(* CoDeSys 2.3 project: cy-wg-019-003.pro *)
(* Title: cy-wg-06 - ClevergyAS *)
(* Author: Andrea Ravasio *)
(* Libraries: Standard.lib 2.12.10 13:48:34, Util.lib 26.9.14 09:12:46, Visual.lib 2.12.10 13:48:34, WagoLibIdent.lib 25.2.13 10:12:16, WagoLibStatus.lib 2.12.10 13:48:32, SysLibFile.lib 2.12.10 13:48:34, SysLibRtc.lib 2.12.10 13:48:32, SysLibSockets.lib 10.2.11 08:20:54, SysLibEvent.lib 2.12.10 13:48:34, SysLibPlcCtrl.lib 2.12.10 13:48:32, SysLibCallback.lib 2.12.10 13:48:32, mod_com.lib 2.12.10 13:48:32, SerComm.lib 31.5.11 07:54:36, Serial_Interface_01.lib 22.4.13 11:50:14, Modb_l05.lib 13.5.15 09:30:08, Ethernet.lib 2.12.10 13:48:32, MBus_03.lib 9.2.13 16:51:58, WagoLibModbus_IP_01.lib 24.7.13 14:05:58, WagoLibMBX_01.lib 20.3.12 15:32:40, LON_01.lib 28.9.12 13:05:10 *)

(* PLC configuration (modules and I/O channels)
VPN_ST2 AT %IX28.0 [BOOLOnX_I] Ch_1 Digital input
LAMP_AL AT %QX18.0 [BOOLOnX_Q] Ch_1 Digital output
KEY_QE_ST AT %IX28.1 [BOOLOnX_I] Ch_2 Digital input
CIR02_EN AT %QX18.1 [BOOLOnX_Q] Ch_2 Digital output
ALARM_PB AT %IX28.2 [BOOLOnX_I] Ch_3 Digital input
CIR01_EN AT %QX18.2 [BOOLOnX_Q] Ch_3 Digital output
CIRD02_A_AL AT %IX28.3 [BOOLOnX_I] Ch_4 Digital input
CIR03_EN AT %QX18.3 [BOOLOnX_Q] Ch_4 Digital output
CIRD02_A_AUTO AT %IX28.4 [BOOLOnX_I] Ch_5 Digital input
AT %QX18.4 [BOOLOnX_Q] Ch_5 Digital output
CIRD02_B_AL AT %IX28.5 [BOOLOnX_I] Ch_6 Digital input
AT %QX18.5 [BOOLOnX_Q] Ch_6 Digital output
CIRD02_B_AUTO AT %IX28.6 [BOOLOnX_I] Ch_7 Digital input
AT %QX18.6 [BOOLOnX_Q] Ch_7 Digital output
CIRD03_A_AL AT %IX28.7 [BOOLOnX_I] Ch_8 Digital input
AT %QX18.7 [BOOLOnX_Q] Ch_8 Digital output
0750-9999/0400-0008 8 DI Generic [Type_1_8_Channels] node 1, in %IB56 out %QB36 {INTTypePAAssignment = PLC; INTTypeModule = plugged}
  CIRD01_B_AUTO AT %IX28.8 [BOOLOnX_I] I 1: Digital Input
  CIR02_ST AT %IX28.9 [BOOLOnX_I] I 2: Digital Input
  CIRD01_A_AL AT %IX28.10 [BOOLOnX_I] I 3: Digital Input
  CIR02_AUTO AT %IX28.11 [BOOLOnX_I] I 4: Digital Input
  CIRD01_A_AUTO AT %IX28.12 [BOOLOnX_I] I 5: Digital Input
  CIR01_AL AT %IX28.13 [BOOLOnX_I] I 6: Digital Input
  CIR02_AL AT %IX28.14 [BOOLOnX_I] I 7: Digital Input
  CIR01_ST AT %IX28.15 [BOOLOnX_I] I 8: Digital Input
0750-9999/0400-0008 8 DI Generic [Type_1_8_Channels] node 2, in %IB57 out %QB37 {INTTypePAAssignment = PLC; INTTypeModule = plugged}
  CIR01_AUTO AT %IX29.0 [BOOLOnX_I] I 1: Digital Input
  CTL03_ST AT %IX29.1 [BOOLOnX_I] I 2: Digital Input
  CIR03_AL AT %IX29.2 [BOOLOnX_I] I 3: Digital Input
  CTL01_ST AT %IX29.3 [BOOLOnX_I] I 4: Digital Input
  CIR03_ST AT %IX29.4 [BOOLOnX_I] I 5: Digital Input
  CTL02_ST AT %IX29.5 [BOOLOnX_I] I 6: Digital Input
  CIR03_AUTO AT %IX29.6 [BOOLOnX_I] I 7: Digital Input
  CIRD01_B_AL AT %IX29.7 [BOOLOnX_I] I 8: Digital Input
0750-9999/0400-0004 4 DI Generic [Type_1_4_Channels] node 3, in %IB58 out %QB37 {INTTypePAAssignment = PLC; INTTypeModule = plugged}
  CIRD03_A_AUTO AT %IX29.8 [BOOLOnX_I] I 1: Digital Input
  CIRD03_B_AUTO AT %IX29.9 [BOOLOnX_I] I 2: Digital Input
  CIRD03_B_AL AT %IX29.10 [BOOLOnX_I] I 3: Digital Input
  AT %IX29.11 [BOOLOnX_I] I 4: Digital Input
0753-0648 LON-FTT [Type_55_1_Channels] node 4, in %IB52 out %QB36 {INTTypePAAssignment = PLC; INTTypeModule = plugged; DataStream = .; DataStream = .; DataStream = .; DataStream = .; DataStream = .; DataStream = .; DataStream = .; DataStream = .; DataStream = .; DataStream = .; DataStream = .; DataStream = .; DataStream = .; DataStream = .; DataStream = .; DataStream = .; DataStream = .; DataStream = .; DataStream = .; DataStream = .; DataStream = .; DataStream = .; DataStream = .; DataStream = .; DataStream = .; DataStream = .; DataStream = .; DataStream = .; DataStream = .; DataStream = .; DataStream = .; DataStream = .; DataStream = .; DataStream = .; DataStream = .; DataStream = .; DataStream = .; DataStream = .; DataStream = .; DataStream = .; DataStream = .; DataStream = .; DataStream = .; DataStream = .; DataStream = .; DataStream = .; DataStream = .; DataStream = .; DataStream = .; DataStream = .; DataStream = .; DataStream = .; DataStream = .; DataStream = .; DataStream = .; DataStream = .; DataStream = .; DataStream = .; DataStream = .; DataStream = .; DataStream = .; DataStream = .; DataStream = .; DataStream = .; DataStream = .; DataStream = .; DataStream = .; DataStream = .; DataStream = .; DataStream = .; DataStream = .; DataStream = .; DataStream = .; DataStream = .; DataStream = .; DataStream = .; DataStream = .; DataStream = .; DataStream = .; DataStream = .; DataStream = .; DataStream = .; DataStream = .; DataStream = .; DataStream = .; DataStream = .; DataStream = .; DataStream = .; DataStream = .; DataStream = .; DataStream = .; DataStream = .; DataStream = .; DataStream = .; DataStream = .; DataStream = .; DataStream = .; DataStream = .; DataStream = .; DataStream = .; DataStream = .; DataStream = .; DataStream = .; DataStream = .; DataStream = .; DataStream = .; DataStream = .; DataStream = .; DataStream = .; DataStream = .; DataStream = .; DataStream = .; DataStream = .; DataStream = .; DataStream = .; DataStream = .; DataStream = .; DataStream = .; DataStream = .; DataStream = .; DataStream = .; DataStream = .; DataStream = .; DataStream = .; DataStream = .; DataStream = .; DataStream = .; DataStream = .; DataStream = .; DataStream = .; DataStream = .; DataStream = .; DataStream = .; DataStream = .; DataStream = .; DataStream = .; DataStream = .; DataStream = .; DataStream = .; DataStream = .; DataStream = .; DataStream = .; DataStream = .; DataStream = .; DataStream = .; DataStream = .; DataStream = .; DataStream = .; DataStream = .; DataStream = .; DataStream = .; DataStream = .; DataStream = .; DataStream = .; DataStream = .; DataStream = .; DataStream = .; DataStream = .; DataStream = .; DataStream = .; DataStream = .; DataStream = .; DataStream = .; DataStream = .; DataStream = .; DataStream = .; DataStream = .; DataStream = .; DataStream = .; DataStream = .; DataStream = .; DataStream = .; DataStream = .; DataStream = .; DataStream = .; DataStream = .; DataStream = .; DataStream = .; DataStream = .; DataStream = .; DataStream = .; DataStream = .; DataStream = .; DataStream = .; DataStream = .; DataStream = .; DataStream = .; DataStream = .; DataStream = .; DataStream = .; DataStream = .; DataStream = .; DataStream = .; DataStream = .; DataStream = .; DataStream = .; DataStream = .; DataStream = .; DataStream = .; DataStream = .}
  AT %IB0 [BYTEOnB_I] First Byte of 24
  AT %QB0 [BYTEOnB_Q] First Byte of 24
0750-0464#04 2/4 AI RTD / ADJ./ HA [Type_44_4_Channels] node 5, in %IB52 out %QB36 {INTTypePAAssignment = PLC; INTTypeModule = plugged}
  S01 AT %IW12 [INTOnW_I] Channel 1
  S02 AT %IW13 [INTOnW_I] Channel 2
  S03 AT %IW14 [INTOnW_I] Channel 3
  S04 AT %IW15 [INTOnW_I] Channel 4
  S05 AT %IW16 [INTOnW_I] Channel 1
  AT %IW17 [INTOnW_I] Channel 2
  S12 AT %IW18 [INTOnW_I] Channel 3
  AT %IW19 [INTOnW_I] Channel 4
0750-0478 2 AI 0-10V 16 Bit S.E. [Type_8_2_Channels] node 7, in %IB84 out %QB60 {INTTypePAAssignment = PLC; INTTypeModule = plugged}
  VRD02_ST AT %IW20 [WORDOnW_I] I 1: Analog Input
  AT %IW21 [WORDOnW_I] I 2: Analog Input
0750-0556 2 AO ±10V [Type_14_2_Channels] node 8, in %IB92 out %QB60 {INTTypePAAssignment = PLC; INTTypeModule = plugged}
  VRD02_CTRL AT %QW12 [WORDOnW_Q] O 1: Analog Output
  AT %QW13 [WORDOnW_Q] O 2: Analog Output
0750-0650/0003-0000#03 RS 232 C Interface (Adjustable), 3 Byte [Type_21_1_Channels] node 9, in %IB96 out %QB60 {INTTypePAAssignment = PLC; INTTypeModule = plugged}
  AT %IX22.0 [BOOLOnX_I] Transmission acknowledgement
  AT %IX22.1 [BOOLOnX_I] Reception request
  AT %IX22.2 [BOOLOnX_I] Initialization acknowledgement
  AT %IX22.3 [BOOLOnX_I] Input buffer is full
  AT %IX22.4 [BOOLOnX_I] Number of received characters Bit 0
  AT %IX22.5 [BOOLOnX_I] Number of received characters Bit 1
  AT %IX22.6 [BOOLOnX_I] Number of received characters Bit 2
  AT %IB45 [BYTEOnB_I] Input data Byte 0
  AT %IB46 [BYTEOnB_I] Input data Byte 1
  AT %IB47 [BYTEOnB_I] Input data Byte 2
  AT %QX14.0 [BOOLOnX_Q] Transmission request
  AT %QX14.1 [BOOLOnX_Q] Reception acknowledgement
  AT %QX14.2 [BOOLOnX_Q] Initialization request
  AT %QX14.4 [BOOLOnX_Q] Number of characters Bit 0
  AT %QX14.5 [BOOLOnX_Q] Number of characters Bit 1
  AT %QX14.6 [BOOLOnX_Q] Number of characters Bit 2
  AT %QB29 [BYTEOnB_Q] Output data Byte 0
  AT %QB30 [BYTEOnB_Q] Output data Byte 1
  AT %QB31 [BYTEOnB_Q] Output data Byte 2
0750-0653/0003-0000#03 RS485 Interface (Adjustable), 3 Bytes [Type_21_1_Channels] node 10, in %IB96 out %QB64 {INTTypePAAssignment = PLC; INTTypeModule = plugged}
  AT %IX24.0 [BOOLOnX_I] Transmission acknowledgement
  AT %IX24.1 [BOOLOnX_I] Reception request
  AT %IX24.2 [BOOLOnX_I] Initialization acknowledgement
  AT %IX24.3 [BOOLOnX_I] Input buffer is full
  AT %IX24.4 [BOOLOnX_I] Number of received characters Bit 0
  AT %IX24.5 [BOOLOnX_I] Number of received characters Bit 1
  AT %IX24.6 [BOOLOnX_I] Number of received characters Bit 2
  AT %IB49 [BYTEOnB_I] Input data Byte 0
  AT %IB50 [BYTEOnB_I] Input data Byte 1
  AT %IB51 [BYTEOnB_I] Input data Byte 2
  AT %QX16.0 [BOOLOnX_Q] Transmission request
  AT %QX16.1 [BOOLOnX_Q] Reception acknowledgement
  AT %QX16.2 [BOOLOnX_Q] Initialization request
  AT %QX16.4 [BOOLOnX_Q] Number of characters Bit 0
  AT %QX16.5 [BOOLOnX_Q] Number of characters Bit 1
  AT %QX16.6 [BOOLOnX_Q] Number of characters Bit 2
  AT %QB33 [BYTEOnB_Q] Output data Byte 0
  AT %QB34 [BYTEOnB_Q] Output data Byte 1
  AT %QB35 [BYTEOnB_Q] Output data Byte 2
0750-0461/0000-0007 2 AI PT100 Resistor Measur. 10R-5k0 [Type_8_2_Channels] node 11, in %IB100 out %QB68 {INTTypePAAssignment = PLC; INTTypeModule = plugged}
  VRD01_ST AT %IW26 [WORDOnW_I] I 1: Analog Input
  AT %IW27 [WORDOnW_I] I 2: Analog Input
VRD01_OP AT %QX18.8 [BOOLOnX_Q] O 1: Digital Output
VRD01_CL AT %QX18.9 [BOOLOnX_Q] O 2: Digital Output
CIRD01_B_EN AT %QX18.10 [BOOLOnX_Q] O 1: Digital Output
CIRD01_A_EN AT %QX18.11 [BOOLOnX_Q] O 2: Digital Output
Fieldbus variables [FB_VARS] node 1, in %IB0 out %QB0
Flag variables [FLAG_VARS] node 2, in %IB0 out %QB0
Modbus-Master [MB_MASTER] node 3, in %IB0 out %QB0
*)

(* Global variable list: Global_Constants *)
VAR_GLOBAL CONSTANT

	Plant_NAME			: STRING :='cySN:19 cyVER:1 - ';
	Plant_SN			: DWORD  :=19;	(* S/N Impianto di telecontrollo *)
	Plant_SW_VER		: WORD   :=1;		(* Versione SW installata *)


	(* Colour defines *)
	COLOR_RED			: DWORD	:= 16#2020F0;
	COLOR_YELLOW		: DWORD	:= 16#20F0F0;
	COLOR_GREEN			: DWORD	:= 16#20F020;
	COLOR_LIGHT_GREEN	: DWORD := 16#006000;

	(* Parameters *)
	Plant_DefaultTAmb	: INT	:=100;		(* [.1°C] Temperatura ambiente di default in caso di rottura sonda *)
	Plant_MaxRunTAmb	: INT   :=210; 		(* [.1°C] Temperatura ambiente massima funzionamento impianto *)
	Plant_AntiFreezeTAmb: INT   :=-40;		(* [.1°C] Antifreeze temperature, start circulators *)
	Plant_VRD_TAlarm	: INT   :=850; 		(* [.1°C] Temperatura di allarme VRD, blocco *)
	Plant_VRD_TMax		: INT   :=800; 		(* [.1°C] Setpoint massimo per uscita VRD *)
	Plant_VRD_TDefault	: INT	:=300;		(* [.1°C] Temperatura di default in caso di errore climatica *)
	Plant_CirOffDelay	: TIME	:=T#30m;	(* (Def.T#15m) Ritardo spegnimento pompe per ricircolo caldaia *)
	Plant_CirOnDelay	: TIME	:=T#15m;
	Plant_MaxWaterLoss	: WORD  :=2;		(* [lt/h] Massima perdita del circuito *)

	(* Filesystem *)
	FilesPath  			: STRING :='S:\';

	(* TCP Logger *)
	Logger_SERVER		: STRING:='';
	Logger_IP			: STRING:='192.168.100.3';
	Logger_PORT			: WORD  :=80;
	Logger_GETSTART		: STRING:='GET /cygmsrv/hsgm.ashx?';
	Logger_GETEND		: STRING:='$R$N$R$N';
	Logger_CHECK		: STRING:='True';
	Logger_CRLF			: STRING:='$R$N';
	Logger_DataFile		: STRING:='S:\LOG.DAT';
	Logger_DataFileOld	: STRING:='S:\LOG.BCK';
	Logger_IndexFile	: STRING:='S:\LOG.IDX';
	Logger_ConnRetries	: BYTE:=5;
	Logger_RecoverMsgs	: BYTE:=25;

	(* TCP Remote *)
	Remote_PORT			: WORD  :=10;
	Remote_WELCOME		: STRING:='Connected$R$N';
	Remote_OK			: STRING:='OK$R$N';
	Remote_ERROR		: STRING:='ERROR$R$N';

	(* TCP Sockets *)
	MAX_SEND_TCP_SERVER					 : DWORD:=3000;(*60000*)
	MAX_RECEIVE_TCP_SERVER				 : DWORD:=3000;
	MAX_RECEIVE_TCP_SERVER_SOCKET	 	 : DWORD:=1500;
	MAX_SEND_TCP_CLIENT					 : DWORD:=3000;(*15000*)
	MAX_RECEIVE_TCP_CLIENT				 : DWORD:=1500;
	MAX_RECEIVE_TCP_CLIENT_SOCKET		 : DWORD:=1500;
	MAX_RECEIVE_UDP_SERVER				 : INT  :=1472;
	MAX_RECEIVE_UDP_CLIENT				 : INT  :=1472;
	CONNECT_WATCHDOG_TIME				 : TIME :=t#10s;

END_VAR


VAR_GLOBAL
	TestNodoInterogato: BYTE;
	NodoDaInterrogare: BYTE;
	InibiscoModbus: BOOL;
END_VAR

(* Global variable list: Global_Retain *)
VAR_GLOBAL RETAIN PERSISTENT
	Mode_Manual : BOOL := FALSE;

	CAL01_Clima : typ_Clima;
	VRD01_Clima : typ_Clima;
	VRD02_Clima : typ_Clima;

	Ctl01_Counter	:	DWORD;	(* Water counter *)
	Ctl02_Counter	:	DWORD;
	Ctl03_Counter	:	DWORD;

	(* Water counter - 2 PULSES/LITER *)
	CTL01	:	obj_CTL	:= (ID:=1, Peso:=10);
	CTL02	:	obj_CTL	:= (ID:=2, Peso:=10);
	CTL03	:	obj_CTL	:= (ID:=3, Peso:=10);


(* Impostazioni di imipanto *)

	DelayAllarmeTemperaturaNonRaggiunta: INT;
	DeltaInterventoAllarmeTempeaturaNonRaggiuta: INT;
	OffsetSetPointManuale:INT;							(* Offset al Setpoint manuale per comensare lo scambiatore *)

	SogliaMinStartAntigelo: INT;
	SogliaMinStopAntigelo: INT;
	BitAbilitaAntigelo: BOOL:=TRUE;

	PercVelMin: INT:=75;
	PercVelMax: INT:=100;
	ErroreTempMax: INT:=100;
	ErroreTempMin: INT:=50;



END_VAR

(* Global variable list: Global_Variables *)
VAR_GLOBAL

	SYS    : typ_SYS;
	Logger : typ_Logger;

	Lamp	:	LAMP_AL_GENERALE;	T_AMB	:	INT;		(* Environment temperature *)

	(**** PLANT OBJECTS ****)
	(*...*)
	(* Boiler *)
	CAL01	:	obj_CAL_VT100GC1B := (ID:=1);


	(* Pumps *)
	(* Single Pumps *)
	CIR01	:	obj_CIR := (ID:=1, CIR_AUTO:=TRUE, OnDelay:=T#1m, OffDelay:=T#30m);
	CIR02	:	obj_CIR := (ID:=2, CIR_AUTO:=TRUE, OnDelay:=T#1m, OffDelay:=T#30m);
	CIR03	:	obj_CIR := (ID:=3, CIR_AUTO:=TRUE, OnDelay:=T#1m, OffDelay:=T#30m);

	(* Double pumps *)
	CIRD01	:	obj_CIR_DOPPIO_new	:= (ID:=1, OnDelay:=T#1m, ExtStatus:=FALSE, Mode:=1);

	(* Modbus Pumps *)
	CIRD02	:	obj_MODBUS_CIR_DOPPIO_DAB := (ID:=1, Address1:=1, Address2:=2, OnDelay:=T#1m, Mode:=1);
	CIRD03	:	obj_MODBUS_CIR_DOPPIO_DAB := (ID:=2, Address1:=3, Address2:=4, OnDelay:=T#1m, Mode:=1);

	(* Valves *)
	VRD01	:	obj_VRD_POT_new	:= (ID:=1, fFeedback:=FALSE,Local_VRD_TAlarm:=800);
	VRD02	:	obj_VRD_new 	:= (ID:=2, fFeedback:=TRUE, ReducedRange := FALSE,Local_VRD_TAlarm:=800);

	(* Temperature probes *)
	TPV01	:	obj_TPV := (ID:=1);
	TPV02	:	obj_TPV := (ID:=2);
	TPV03	:	obj_TPV := (ID:=3);
	TPV04	:	obj_TPV := (ID:=4);
	TPV05	:	obj_TPV := (ID:=5);
	TPV12	:	obj_TPV := (ID:=6);

	(* ZigBee temperature probes *)
	ZTHL06	:	obj_ZTHL := (ID:=1, Address:=11);   	(* Ala nuova Fan Coil *)
	ZTHL07	:	obj_ZTHL := (ID:=2, Address:=12);	(* Ala nuova Fan Coil *)
	ZTHL08	:	obj_ZTHL := (ID:=3, Address:=13);	(* Ala vecchia Radiatori *)
	ZTHL09	:	obj_ZTHL := (ID:=4, Address:=14);	(* Ala vecchia Radiatori *)
	ZTHL10	:	obj_ZTHL := (ID:=5, Address:=15);	(* Palestra Fan Coil *)
(*	ZTHL11	:	obj_ZTHL := (ID:=6, Address:=6); *)

	(* Heat recorders *)
	CTB01	:	obj_MBUS_CTB_SHARKY775 := (ID:=1, Address:=16#49881918);
	CTB02	:	obj_MBUS_CTB_SHARKY775 := (ID:=2, Address:=16#51867410);	(* Non collegato *)

	(* Cronothermostat *)
	THER01	:	obj_CRONTER_01:= (ID:=1, Local_MaxRunTAmb:=250,Histeresys:=10);
	THER02	:	obj_CRONTER_01 := (ID:=2, Local_MaxRunTAmb:=250,Histeresys:=10);
	THER03	:	obj_CRONTER_01 := (ID:=3, Local_MaxRunTAmb:=250,Histeresys:=10);
	THER04	:	obj_CRONTER_01 := (ID:=4, Local_MaxRunTAmb:=800,Histeresys:=10);
	THER05	:	obj_CRONTER_01 := (ID:=5, Local_MaxRunTAmb:=800,Histeresys:=10);
	THER06	:	obj_CRONTER_01 := (ID:=6, Local_MaxRunTAmb:=800,Histeresys:=10);
	THER250	:	obj_CRONTER_01 := (ID:=250, Local_MaxRunTAmb:=250,Histeresys:=10);

	CronEd	: obj_CRON_EDITOR_01;

	(** Communication **)
	(* ModBus *)
	MODB01	:	obj_MODBUS		:= (ID:=1, COM:=3, BAUDRATE:=BAUD_19200, RS485:=TRUE);
	MODB02	:	obj_MODBUS_TCP 	:= (ID:=1, IP:='192.168.100.4');

	(* M-Bus *)
	MBUS01	:	obj_MBUS		:= (ID:=1, COM:=2, BAUDRATE:=BAUD_2400);

	(**** SIMULATION ONLY ****)
	(*...*)
END_VAR

(* Global variable list: LON/Module_1/InterfaceBlock_Module_1 *)
VAR_GLOBAL CONSTANT
(******************************************)
(* Automatic generated code, do not edit! *)
(******************************************)
	abSignature_Module_1 : ARRAY[0..15] OF BYTE := 16#0B,16#F9,16#43,16#24,16#44,16#59,16#3B,16#4F,16#A3,16#F7,16#62,16#F6,16#7A,16#4E,16#21,16#9A;
	wConfigSize_Module_1 : WORD := 522;
	abInterface_Module_1 : ARRAY[0..130] OF DWORD :=
		16#302841AA, 16#2113D509, 16#6041B800, 16#06246830, 16#428B2E71, 16#64B95263, 16#FE000902, 16#2A050140, 
		16#0028C092, 16#037C10FF, 16#6D81026F, 16#0418B0E4, 16#C75C1D07, 16#9CD47157, 16#5A1D2B75, 16#1D531D1E, 
		16#4F0D2658, 16#5AC76C1D, 16#2D5F874A, 16#FE884D09, 16#CE34C958, 16#4CA0345D, 16#856A742A, 16#B26FDD52, 
		16#2BF66959, 16#74C79655, 16#966CD09D, 16#DFE60549, 16#2C48B975, 16#B66DFB76, 16#48BA6ECB, 16#955B162D, 
		16#B7300196, 16#2B35AD5D, 16#65EBC62D, 16#2106DDB9, 16#564CBE30, 16#DDA96F05, 16#AD4B372C, 16#255378CD, 
		16#36ADD181, 16#59D42ACB, 16#9B603585, 16#DDC49858, 16#EA45B329, 16#CD59F616, 16#B50A12E0, 16#56B5BE52, 
		16#8C890100, 16#5AAA1481, 16#B253E154, 16#6C831684, 16#A2ADDCB0, 16#4ABD13A9, 16#950B79D9, 16#4A948694, 
		16#4DBF5E45, 16#CA018948, 16#054C41E5, 16#B86DCB52, 16#2FBEA018, 16#40AAB4D0, 16#A1F866E7, 16#E288A8D1, 
		16#D192DBA2, 16#80E25047, 16#84B4644B, 16#B225A097, 16#59A9F8AC, 16#2D5B376E, 16#7B32E9CE, 16#B7AE3099, 
		16#2D551A30, 16#03F1D236, 16#C96176D0, 16#D94ABD0C, 16#94950479, 16#60B2886A, 16#25C9C990, 16#4CBCB141, 
		16#32D60DA9, 16#6A1D86D9, 16#514404B2, 16#129278D2, 16#09A12969, 16#AB6529E7, 16#90EE2F05, 16#10604094, 
		16#FE031C08, 16#418817F3, 16#84320FB0, 16#238F21C0, 16#6F23C08A, 16#003E98A3, 16#80677304, 16#10728E02, 
		16#0E02FC59, 16#02343A1A, 16#183B223A, 16#804705C0, 16#47864080, 16#47408082, 16#2E208347, 16#A304A014, 
		16#121794C3, 16#81595C58, 16#C785A471, 16#6820171C, 16#7201925C, 16#88CB8581, 16#5D283A17, 16#2378C120, 
		16#1724EF85, 16#0B5F78C0, 16#85687C01, 16#CE17B4F2, 16#814B5FD8, 16#F6856C7D, 16#E8DC173C, 16#6001805F, 
		16#047C0101, 16#97310112, 16#A061674C, 16#20841212, 16#4081A022, 16#CDBF90E0, 16#AC44490E, 16#3FFAE9CE, 
		16#7AED8BBD, 16#5F7348A7, 16#0000304C;
END_VAR

(* Global variable list: LON/Module_2/InterfaceBlock_Module_2 *)
VAR_GLOBAL CONSTANT
(******************************************)
(* Automatic generated code, do not edit! *)
(******************************************)
	abSignature_Module_2 : ARRAY[0..15] OF BYTE := 16#A8,16#5E,16#16,16#AC,16#64,16#CD,16#36,16#4E,16#96,16#14,16#FA,16#F3,16#A9,16#72,16#20,16#9F;
	wConfigSize_Module_2 : WORD := 522;
	abInterface_Module_2 : ARRAY[0..130] OF DWORD :=
		16#302841AA, 16#21F36F08, 16#6041B800, 16#06246830, 16#428B2E71, 16#64B95263, 16#FE000902, 16#2A050140, 
		16#0028C092, 16#037C10FF, 16#6D81026F, 16#0418B0E4, 16#C75C1D07, 16#9CD47157, 16#5A1D2B75, 16#1D531D1E, 
		16#4F0D2658, 16#5AC76C1D, 16#2D5F874A, 16#FE884D09, 16#CE34C958, 16#4CA0345D, 16#856A742A, 16#B26FDD52, 
		16#2BF66959, 16#74C79655, 16#966CD09D, 16#DFE60549, 16#2C48B975, 16#B66DFB76, 16#48BA6ECB, 16#955B162D, 
		16#B7300196, 16#2B35AD5D, 16#65EBC62D, 16#2106DDB9, 16#564CBE30, 16#DDA96F05, 16#AD4B372C, 16#255378CD, 
		16#36ADD181, 16#59D42ACB, 16#9B603585, 16#DDC49858, 16#EA45B329, 16#CD59F616, 16#B50A12E0, 16#56B5BE52, 
		16#8C890100, 16#5AAA1481, 16#B253E154, 16#6C831684, 16#A2ADDCB0, 16#4ABD13A9, 16#950B79D9, 16#4A948694, 
		16#4DBF5E45, 16#CA018948, 16#054C41E5, 16#B86DCB52, 16#2FBEA018, 16#40AAB4D0, 16#A1F866E7, 16#E288A8D1, 
		16#D192DBA2, 16#80E25047, 16#84B4644B, 16#B225A097, 16#59A9F8AC, 16#2D5B376E, 16#7B32E9CE, 16#B7AE3099, 
		16#2D551A30, 16#03F1D236, 16#C96176D0, 16#D94ABD0C, 16#94950479, 16#60B2886A, 16#25C9C990, 16#4CBCB141, 
		16#32D60DA9, 16#6A1D86D9, 16#514404B2, 16#129278D2, 16#09A12969, 16#AB6529E7, 16#90EE2F05, 16#10604094, 
		16#FE031C08, 16#418817F3, 16#84320FB0, 16#238F21C0, 16#6F23C08A, 16#003E98A3, 16#80677304, 16#10728E02, 
		16#0E02FC59, 16#02343A1A, 16#183B223A, 16#804705C0, 16#47864080, 16#47408082, 16#2E208347, 16#A304A014, 
		16#121794C3, 16#81595C58, 16#C785A471, 16#6820171C, 16#7201925C, 16#88CB8581, 16#5D283A17, 16#2378C120, 
		16#1724EF85, 16#0B5F78C0, 16#85687C01, 16#CE17B4F2, 16#814B5FD8, 16#F6856C7D, 16#E8DC173C, 16#6001805F, 
		16#047C0101, 16#97310112, 16#A061674C, 16#20841212, 16#4081A022, 16#F48A9AE0, 16#E664595B, 16#68D9A9CD, 
		16#A9E7EBA7, 16#FC3348B9, 16#000088AD;
END_VAR

(* Global variable list: LON/Module_1/Runtime_Module_1 *)
VAR_GLOBAL
(******************************************)
(* Automatic generated code, do not edit! *)
(******************************************)
	mbxModule_1 : MBX_Full;
	InDataTelegram_Module_1 : ARRAY[0..255] OF BYTE;
	OutDataTelegram_Module_1 : ARRAY[0..511] OF BYTE;

	xInitRunning_Module_1 : BOOL := FALSE;
	unLastLen_mbxModule_1 : UINT;
END_VAR

(* Global variable list: LON/Module_2/Runtime_Module_2 *)
VAR_GLOBAL
(******************************************)
(* Automatic generated code, do not edit! *)
(******************************************)
	mbxModule_2 : MBX_Full;
	InDataTelegram_Module_2 : ARRAY[0..255] OF BYTE;
	OutDataTelegram_Module_2 : ARRAY[0..511] OF BYTE;

	xInitRunning_Module_2 : BOOL := FALSE;
	unLastLen_mbxModule_2 : UINT;
END_VAR

(* Data type in LON/Enumerations *)
TYPE alarm_type_t :
(
	AL_HEADER := -13,
	AL_FOOTER := -12,
	AL_DEBUG := -11,
	AL_INFO := -10,
	AL_SYSTEM_INFO := -6,
	AL_VALUE_INVALID := -5,
	AL_CONSTANT := -4,
	AL_OFFLINE := -3,
	AL_UNKNOWN := -2,
	AL_NUL := -1,
	AL_NO_CONDITION := 0,
	AL_ALM_CONDITION := 1,
	AL_TOT_SVC_ALM_1 := 2,
	AL_TOT_SVC_ALM_2 := 3,
	AL_TOT_SVC_ALM_3 := 4,
	AL_LOW_LMT_CLR_1 := 5,
	AL_LOW_LMT_CLR_2 := 6,
	AL_HIGH_LMT_CLR_1 := 7,
	AL_HIGH_LMT_CLR_2 := 8,
	AL_LOW_LMT_ALM_1 := 9,
	AL_LOW_LMT_ALM_2 := 10,
	AL_HIGH_LMT_ALM_1 := 11,
	AL_HIGH_LMT_ALM_2 := 12,
	AL_FIR_ALM := 13,
	AL_FIR_PRE_ALM := 14,
	AL_FIR_TRBL := 15,
	AL_FIR_SUPV := 16,
	AL_FIR_TEST_ALM := 17,
	AL_FIR_TEST_PRE_ALM := 18,
	AL_FIR_ENVCOMP_MAX := 19,
	AL_FIR_MONITOR_COND := 20,
	AL_FIR_MAINT_ALERT := 21,
	AL_FATAL_ERROR := 30,
	AL_ERROR := 31,
	AL_WARNING := 32
);
END_TYPE

(* Data type in Logger *)
TYPE en_Logger_ErrLev :
(
	EL_Log			:=0,
	EL_Wrn			:=1,
	EL_Alarm		:=2,
	EL_AlarmStop	:=3
);
END_TYPE

(* Data type in Logger *)
TYPE en_Logger_Status :
(
	S_Logger_UNKNOWN := 0,
	S_Logger_IDLE,
	S_Logger_WAITCONN,
	S_Logger_WAITTX,
	S_Logger_WAITRESP,
	S_Logger_ERROR
);
END_TYPE

(* Data type *)
TYPE en_SYS_Objects :
(
	EO_SYS		:=0,  (* PLC *)
	EO_VPN		:=1,  (* VPN *)
	EO_DOOR		:=2,  (* Door & access control *)

	EO_CAL		:=10, (* Caldaia *)
	EO_CIR		:=11, (* Circolatore *)
	EO_CRON		:=12, (* Crono-termostato *)
	EO_VRD		:=13, (* Valvola miscelatore pannelli *)
	EO_CTL		:=14, (* Contalitri *)
	EO_CTB		:=15, (* Contabilizzatore *)
	EO_TPV		:=16, (* Temperature probes values *)
	EO_PPV		:=17, (* Pressure probes values *)
	EO_PBV		:=18, (* Over-Pressure Alarms *)
	EO_TBV		:=19, (* Over-Temperature Alarms *)
	EO_PMV		:=20, (* Under-Pressure Alarms *)
	EO_GRU		:=21, (* Gruppo termico *)
	EO_PDC		:=22, (* Pompa di calore *)
	EO_SOL		:=23, (* Pannello solare termico *)
	EO_ESOL		:=24, (* Pannello solare fotovoltaico *)
	EO_GAS		:=25, (* Contatore GAS *)
	EO_PORT		:=26, (* Misuratore di portata *)
	EO_FPV		:=27, (* Flow probes values *)
	EO_ANZ		:=28, (* Analizzatore di rete *)
	EO_SCA		:=29, (* Signal Control Alarms *)
	EO_LUX		:=30, (* Base Illumination point *)
	EO_LUXM		:=31, (* Metered Illumination point *)
	EO_PSG		:=32, (* Sensore di passaggio *)
	EO_HVAC		:=33, (* Heating, Ventilating and Air Conditioning *)
	EO_HYGRV	:=34, (* Relative Humidity sensors value *)
	EO_COOV		:=35, (* Carbon Dioxide CO2 sensors value *)
	EO_INV		:=36, (* Inverter *)
	EO_STR		:=37, (* Smart string box *)

	EO_CIRD		:=39, (* Double CIR *)
	EO_ACS		:=40, (* Hot domestic water *)
	EO_FRG		:=41, (* Frigo *)
	EO_THER		:=42, (* Thermostat *)
	EO_CIRM		:=43, (* Modbus CIR *)
	EO_CIRDM	:=44, (* Modbus double CIR *)

	EO_ZGW			:=200,  (* ZigBee - Gateway *)
	EO_ZRM			:=201,	(* ZigBee - Repeater *)
	EO_ZREL			:=202,	(* ZigBee - Actuator rele *)
	EO_ZTHL			:=203,	(* ZigBee - Temperature Sensor *)

	EO_ASGW			:=250,	(* ASi - Gateway *)
	EO_ASCBI		:=251,	(* ASi - Input Board, Ciabatta *)

	EO_LON			:=1000, (* Bus - LON *)
	EO_MODBUS		:=1001, (* Bus - MODBUS *)
	EO_MBUS			:=1002, (* Bus - M-BUS *)
	EO_MODBUS_TCP	:=1003, (* Bus - MODBUS TCP *)

	EO_GENERIC		:=9000, (* Generic dataset *)
	EO_EXPO			:=9001 (* EXPO dataset *)
);
END_TYPE

(* Data type *)
TYPE en_SYS_Status :
(
	S_UNKNOWN  := 0,
	S_STARTUP,
	S_INIT_RTC,
	S_INIT_VAR,
	S_AUTOTEST,
	S_RUNNING,
	S_SHUTDOWN,
	S_HALT
);
END_TYPE

(* Data type in LON/Enumerations *)
TYPE file_request_t :
(
	FR_NUL := -1,
	FR_OPEN_TO_SEND := 0,
	FR_OPEN_TO_RECEIVE := 1,
	FR_CLOSE_FILE := 2,
	FR_CLOSE_DELETE_FILE := 3,
	FR_DIRECTORY_LOOKUP := 4,
	FR_OPEN_TO_SEND_RA := 5,
	FR_OPEN_TO_RECEIVE_RA := 6
);
END_TYPE

(* Data type in LON/Enumerations *)
TYPE file_status_t :
(
	FS_NUL := -1,
	FS_XFER_OK := 0,
	FS_LOOKUP_OK := 1,
	FS_OPEN_FAIL := 2,
	FS_LOOKUP_ERR := 3,
	FS_XFER_UNDERWAY := 4,
	FS_IO_ERR := 5,
	FS_TIMEOUT_ERR := 6,
	FS_WINDOW_ERR := 7,
	FS_AUTH_ERR := 8,
	FS_ACCESS_UNAVAIL := 9,
	FS_SEEK_INVALID := 10,
	FS_SEEK_WAIT := 11
);
END_TYPE

(* Data type in LON/Enumerations *)
TYPE hvac_t :
(
	HVAC_NUL := -1,
	HVAC_AUTO := 0,
	HVAC_HEAT := 1,
	HVAC_MRNG_WRMUP := 2,
	HVAC_COOL := 3,
	HVAC_NIGHT_PURGE := 4,
	HVAC_PRE_COOL := 5,
	HVAC_OFF := 6,
	HVAC_TEST := 7,
	HVAC_EMERG_HEAT := 8,
	HVAC_FAN_ONLY := 9,
	HVAC_FREE_COOL := 10,
	HVAC_ICE := 11,
	HVAC_MAX_HEAT := 12,
	HVAC_ECONOMY := 13,
	HVAC_DEHUMID := 14,
	HVAC_CALIBRATE := 15,
	HVAC_EMERG_COOL := 16,
	HVAC_EMERG_STEAM := 17,
	HVAC_MAX_COOL := 18,
	HVAC_HVC_LOAD := 19,
	HVAC_NO_LOAD := 20
);
END_TYPE

(* Data type in LON/Enumerations *)
TYPE object_request_t :
(
	RQ_NUL := -1,
	RQ_NORMAL := 0,
	RQ_DISABLED := 1,
	RQ_UPDATE_STATUS := 2,
	RQ_SELF_TEST := 3,
	RQ_UPDATE_ALARM := 4,
	RQ_REPORT_MASK := 5,
	RQ_OVERRIDE := 6,
	RQ_ENABLE := 7,
	RQ_RMV_OVERRIDE := 8,
	RQ_CLEAR_STATUS := 9,
	RQ_CLEAR_ALARM := 10,
	RQ_ALARM_NOTIFY_ENABLED := 11,
	RQ_ALARM_NOTIFY_DISABLED := 12,
	RQ_MANUAL_CTRL := 13,
	RQ_REMOTE_CTRL := 14,
	RQ_PROGRAM := 15,
	RQ_CLEAR_RESET := 16,
	RQ_RESET := 17,
	RQ_CLEAR_LOG := 18,
	RQ_LOAD_PROGRAM := 19,
	RQ_RUN_PROGRAM := 20,
	RQ_HALT_PROGRAM := 21,
	RQ_RESTART_PROGRAM := 22,
	RQ_UNLOAD_PROGRAM := 23,
	RQ_STEP_PROGRAM := 24
);
END_TYPE

(* Data type in LON/Enumerations *)
TYPE priority_level_t :
(
	PR_NUL := -1,
	PR_LEVEL_0 := 0,
	PR_LEVEL_1 := 1,
	PR_LEVEL_2 := 2,
	PR_LEVEL_3 := 3,
	PR_1 := 4,
	PR_2 := 5,
	PR_3 := 6,
	PR_4 := 7,
	PR_6 := 8,
	PR_8 := 9,
	PR_10 := 10,
	PR_16 := 11
);
END_TYPE

(* Data type in Plant_Objects *)
TYPE typ_Clima : (* CURVA CLIMATICA *)
STRUCT
	InitOK:		BOOL;
	Points: 	ARRAY [0..10] OF POINT;
END_STRUCT
END_TYPE

(* Data type in Plant_Objects *)
TYPE typ_Cron_Calendar :
STRUCT
	Profile		: ARRAY[0..384] OF BYTE;
END_STRUCT
END_TYPE

(* Data type in Plant_Objects *)
TYPE typ_Cron_Jolly :
STRUCT
	Start		: DT;
	End			: DT;
	Temp		: WORD;
	Flags		: WORD; (* B0:Enabled B1..B15:Unused *)
END_STRUCT
END_TYPE

(* Data type in Plant_Objects *)
TYPE typ_Cron_Profile :
STRUCT
	Flags		: WORD;
	Setpoint	: ARRAY [0..95] OF WORD;
END_STRUCT
END_TYPE

(* Data type in Logger *)
TYPE typ_Logger :
STRUCT
	Status		: en_Logger_Status;

	SendReq		: BOOL;
	SendIdx		: DWORD;
	SendData	: ARRAY [0..MAX_SEND_TCP_CLIENT] OF BYTE;
	SendLen		: DINT;

	TData		: ARRAY [0..MAX_SEND_TCP_CLIENT] OF BYTE;
	TLen		: DINT;

	LastIdxPos	: DWORD;

	(* Temporary variables used by objects *)
	s1			: STRING(256);
	i1			: WORD;

END_STRUCT
END_TYPE

(* Data type in Plant_Objects *)
TYPE typ_MODBUS_ABB_DMTME72 :
STRUCT
	V_3P		: DWORD; (* V *)
	V_L1N		: DWORD;
	V_L2N		: DWORD;
	V_L3N		: DWORD;
	V_L1L2		: DWORD;
	V_L2L3		: DWORD;
	V_L3L1		: DWORD;
	I_3P		: DWORD; (* 10^-3 A *)
	I_L1		: DWORD;
	I_L2		: DWORD;
	I_L3		: DWORD;
	PF_3P		: DINT;	 (* 10^-3 *)
	PF_L1		: DINT;
	PF_L2		: DINT;
	PF_L3		: DINT;
	COS_3P		: DINT;  (*NO!*)
	COS_L1		: DINT;
	COS_L2		: DINT;
	COS_L3		: DINT;
	VA_3P		: DWORD; (* VA *)(*NO!*)
	VA_L1		: DWORD;
	VA_L2		: DWORD;
	VA_L3		: DWORD;
	P_3P		: DWORD; (* W *)
	P_L1		: DWORD;
	P_L2		: DWORD;
	P_L3		: DWORD;
	Q_3P		: DWORD; (* VAr *)
	Q_L1		: DWORD;
	Q_L2		: DWORD;
	Q_L3		: DWORD;

	WH_3P		: DWORD; (* 10^-1 kWh *)
	VARH_3P		: DWORD; (* 10^-1 kVArh *)
	FREQ		: DWORD; (* 10^-3 Hz *)

	I_L1_Max	: DWORD;
	I_L2_Max	: DWORD;
	I_L3_Max	: DWORD;
	P_3P_Max	: DWORD;
	Q_3P_Max	: DWORD;
	P_3P_Avg15m	: DWORD;

END_STRUCT
END_TYPE

(* Data type in Plant_Objects *)
TYPE typ_MODBUS_CIR :
STRUCT
	PumpStatus		:	WORD;
	PumpFault		:	BOOL;
	PumpBoardTemp	:	INT;	(* Electonic board temperature  [°C] *)
	PumpVoltage		:	WORD;	(* Input voltage rms [V] *)
	PumpCurrent		:	WORD;	(* Output current [E-3 A]	*)
	PumpRPM			:	WORD;	(* Round per minute [rpm] *)
	PumpPower		:	WORD;	(* Power [W] *)
	PumpOpTime		:	DWORD;	(* Pump operating time [h] *)
	PumpHead		:	WORD;	(* [E-1 m] *)
	PumpFlow		:	WORD;	(* Extimated flow [E-1 m3/h] *)
	PumpLiqTemp		:	WORD;	(* Liquid temperature [°C] *)
	PumpAlarm		:	ARRAY [0..14] OF WORD;

END_STRUCT
END_TYPE

(* Data type in Plant_Objects *)
TYPE typ_MODBUS_ELGAS_MINIELCOR :
STRUCT
	Vb			: ARRAY [0..3] OF WORD;	(* m^3 *)
	Vm			: DWORD;				(* m^3 *)
	P			: REAL;					(* bar *)
	T			: REAL;					(* °C *)
	C			: REAL;
	Vbs			: ARRAY [0..3] OF WORD;	(* m^3 *)
	Vb_d_d		: ARRAY [0..3] OF WORD;	(* m^3 *)
	Vb_d_m		: ARRAY [0..3] OF WORD;	(* m^3 *)
	Vm_d_d		: DWORD;				(* m^3 *)
	Q			: REAL;					(* m^3/h *)
	Qb			: REAL;					(* m^3/h *)

	BC_EVC		: REAL;			(* % *)
	BV_EVC		: REAL;			(* V *)
	D_Err		: WORD;			(* 0:OK, 1:FAIL *)
	Status		: DWORD;		(* Status bits *)

END_STRUCT
END_TYPE

(* Data type in Plant_Objects *)
TYPE typ_MODBUS_FRER_IQ96U2 :
STRUCT
	V_L1N		: DWORD; (* 10^-3 V *)
	V_L2N		: DWORD;
	V_L3N		: DWORD;
	V_L1L2		: DWORD;
	V_L2L3		: DWORD;
	V_L3L1		: DWORD;
	I_L1		: DWORD; (* 10^-3 I *)
	I_L2		: DWORD;
	I_L3		: DWORD;
	FREQ		: DWORD; (* 10^-3 Hz *)
	P_3P		: DWORD; (* W *)
	Q_3P		: DWORD; (* VAr *)
	PF_3P		: DINT;	 (* 10^-3 *)
	WH_3P		: DWORD; (* Wh *)
	VARH_3P		: DWORD; (* VArh *)
	MULT		: DWORD;

	WH_3P_NEG	: DWORD; (* Wh *)
	VARH_3P_NEG : DWORD; (* VArh *)
	S_3P		: DWORD; (* VA *)

	PF_L1		: DWORD; (* 10^-3 *)
	PF_L2		: DWORD; (* 10^-3 *)
	PF_L3		: DWORD; (* 10^-3 *)

	P_3P_Max	: DWORD;
	P_3P_Avg15m	: DWORD;
	I_L1_Max	: DWORD;
	I_L2_Max	: DWORD;
	I_L3_Max	: DWORD;
	I_L1_Avg15m	: DWORD;
	I_L2_Avg15m	: DWORD;
	I_L3_Avg15m	: DWORD;

END_STRUCT
END_TYPE

(* Data type in Plant_Objects *)
TYPE typ_MODBUS_VAR : (* Gestione parametri MODBUS *)
STRUCT
	SlaveAddress	: BYTE;
	FunCode			: BYTE;
	FunAddress		: WORD;
	Refresh_Time	: BYTE; (* 0:No refresh x:Refresh in seconds *)
	Refresh_Cnt		: BYTE; (* INTERNAL *)
	Variable		: POINTER TO WORD;
	Variable_Size	: BYTE;
	Variable_Mirror : WORD; (* INTERNAL [Force refresh on read variables when <>0] *)
END_STRUCT
END_TYPE

(* Data type *)
TYPE typ_SYS :
STRUCT
	Status			: en_SYS_Status;
	Warning			: BOOL;
	Alarm			: BOOL;
	AlarmStop		: BOOL;

	Time_LogString	: STRING;
	Time_Year		: WORD;
	Time_Month		: BYTE;
	Time_Day		: BYTE;
	Time_Hour		: BYTE;
	Time_Minute		: BYTE;

	Time_CT_DT		: DT;
	Time_CT_Day		: WORD;
	Time_CT_Quarter	: BYTE;

	LastLogs_Idx	: BYTE;
	LastLogs_Dat	: ARRAY[0..5] OF STRING;
	LastLogs_Msg	: ARRAY[0..5] OF STRING;

END_STRUCT
END_TYPE

(* Data type in Plant_Objects *)
TYPE typ_VisuStrutturaMbus :
STRUCT

	sdNodoPresente: STRING(16);
	sdEnergia: STRING(16);
	sdPotenza: STRING(16);
	sdVolume: STRING(16);
	sdFlow: STRING(16);
	sdTempIngresso: STRING(8);
	sdTempaUscita: STRING(8);
	sdTempDelta: STRING(8);

END_STRUCT
END_TYPE

(* Data type in LON/NetworkVariables *)
TYPE typSnvtAlarm : 
STRUCT
	abLocation : ARRAY[0..5] OF BYTE;
	wObjectId : WORD;
	bAlarmType : BYTE (* enum type alarm_type_t *);
	bPriorityLevel : BYTE (* enum type priority_level_t *);
	wIndexToSnvt : WORD;
	abValue : ARRAY[0..3] OF BYTE;
	wYear : WORD;
	bMonth : BYTE;
	bDay : BYTE;
	bHour : BYTE;
	bMinute : BYTE;
	bSecond : BYTE;
	wMillisecond : WORD;
	abAlarmLimit : ARRAY[0..3] OF BYTE;
	bStatusInformation : BYTE; (* bit allocation of bStatusInformation:
	bit 0: NVI update counter LSB
	bit 1: NVI update counter
	bit 2: NVI update counter
	bit 3: NVI update counter MSB
	bit 4: timeout for NVI occurs (MaxRcvTime expired)
	bit 5: reserved
	bit 6: reserved
	bit 7: force NVO update *)
	bInternalUseOnly : BYTE; (* Do not use this byte in your application! *)
END_STRUCT
END_TYPE

(* Data type in LON/NetworkVariables *)
TYPE typSnvtFilePos : 
STRUCT
	diRwPtr : DINT;
	wRwLength : WORD;
	bStatusInformation : BYTE; (* bit allocation of bStatusInformation:
	bit 0: NVI update counter LSB
	bit 1: NVI update counter
	bit 2: NVI update counter
	bit 3: NVI update counter MSB
	bit 4: timeout for NVI occurs (MaxRcvTime expired)
	bit 5: reserved
	bit 6: reserved
	bit 7: force NVO update *)
	bInternalUseOnly : BYTE; (* Do not use this byte in your application! *)
END_STRUCT
END_TYPE

(* Data type in LON/NetworkVariables *)
TYPE typSnvtFileReq : 
STRUCT
	bRequest : BYTE (* enum type file_request_t *);
	wIndex : WORD;
	wReceiveTimeout : WORD;
	abDestAddress : ARRAY[0..4] OF BYTE (* union declaration *);
	bAuthOn : BYTE;
	bPrioOn : BYTE;
	bStatusInformation : BYTE; (* bit allocation of bStatusInformation:
	bit 0: NVI update counter LSB
	bit 1: NVI update counter
	bit 2: NVI update counter
	bit 3: NVI update counter MSB
	bit 4: timeout for NVI occurs (MaxRcvTime expired)
	bit 5: reserved
	bit 6: reserved
	bit 7: force NVO update *)
	bInternalUseOnly : BYTE; (* Do not use this byte in your application! *)
END_STRUCT
END_TYPE

(* Data type in LON/NetworkVariables *)
TYPE typSnvtFileStatus : 
STRUCT
	bStatus : BYTE (* enum type file_status_t *);
	wNumberOfFiles : WORD;
	wSelectedFile : WORD;
	abAdr : ARRAY[0..21] OF BYTE (* union declaration *);
	bStatusInformation : BYTE; (* bit allocation of bStatusInformation:
	bit 0: NVI update counter LSB
	bit 1: NVI update counter
	bit 2: NVI update counter
	bit 3: NVI update counter MSB
	bit 4: timeout for NVI occurs (MaxRcvTime expired)
	bit 5: reserved
	bit 6: reserved
	bit 7: force NVO update *)
	bInternalUseOnly : BYTE; (* Do not use this byte in your application! *)
END_STRUCT
END_TYPE

(* Data type in LON/NetworkVariables *)
TYPE typSnvtHvacMode : 
STRUCT
	bSnvtHvacMode : BYTE (* enum type hvac_t *);
	bStatusInformation : BYTE; (* bit allocation of bStatusInformation:
	bit 0: NVI update counter LSB
	bit 1: NVI update counter
	bit 2: NVI update counter
	bit 3: NVI update counter MSB
	bit 4: timeout for NVI occurs (MaxRcvTime expired)
	bit 5: reserved
	bit 6: reserved
	bit 7: force NVO update *)
	bInternalUseOnly : BYTE; (* Do not use this byte in your application! *)
END_STRUCT
END_TYPE

(* Data type in LON/NetworkVariables *)
TYPE typSnvtObjRequest : 
STRUCT
	wObjectId : WORD;
	bObjectRequest : BYTE (* enum type object_request_t *);
	bStatusInformation : BYTE; (* bit allocation of bStatusInformation:
	bit 0: NVI update counter LSB
	bit 1: NVI update counter
	bit 2: NVI update counter
	bit 3: NVI update counter MSB
	bit 4: timeout for NVI occurs (MaxRcvTime expired)
	bit 5: reserved
	bit 6: reserved
	bit 7: force NVO update *)
	bInternalUseOnly : BYTE; (* Do not use this byte in your application! *)
END_STRUCT
END_TYPE

(* Data type in LON/NetworkVariables *)
TYPE typSnvtObjStatus : 
STRUCT
	wObjectId : WORD;
	bBitfieldByteOffset2 : BYTE (* bit field *);
	bBitfieldByteOffset3 : BYTE (* bit field *);
	bBitfieldByteOffset4 : BYTE (* bit field *);
	bBitfieldByteOffset5 : BYTE (* bit field *);
	bStatusInformation : BYTE; (* bit allocation of bStatusInformation:
	bit 0: NVI update counter LSB
	bit 1: NVI update counter
	bit 2: NVI update counter
	bit 3: NVI update counter MSB
	bit 4: timeout for NVI occurs (MaxRcvTime expired)
	bit 5: reserved
	bit 6: reserved
	bit 7: force NVO update *)
	bInternalUseOnly : BYTE; (* Do not use this byte in your application! *)
END_STRUCT
END_TYPE

(* Data type in LON/NetworkVariables *)
TYPE typSnvtState : 
STRUCT
	bBitfieldByteOffset0 : BYTE (* bit field *);
	bBitfieldByteOffset1 : BYTE (* bit field *);
	bStatusInformation : BYTE; (* bit allocation of bStatusInformation:
	bit 0: NVI update counter LSB
	bit 1: NVI update counter
	bit 2: NVI update counter
	bit 3: NVI update counter MSB
	bit 4: timeout for NVI occurs (MaxRcvTime expired)
	bit 5: reserved
	bit 6: reserved
	bit 7: force NVO update *)
	bInternalUseOnly : BYTE; (* Do not use this byte in your application! *)
END_STRUCT
END_TYPE

(* Data type in LON/NetworkVariables *)
TYPE typSnvtSwitch : 
STRUCT
	bValue : BYTE;
	siState : SINT;
	bStatusInformation : BYTE; (* bit allocation of bStatusInformation:
	bit 0: NVI update counter LSB
	bit 1: NVI update counter
	bit 2: NVI update counter
	bit 3: NVI update counter MSB
	bit 4: timeout for NVI occurs (MaxRcvTime expired)
	bit 5: reserved
	bit 6: reserved
	bit 7: force NVO update *)
	bInternalUseOnly : BYTE; (* Do not use this byte in your application! *)
END_STRUCT
END_TYPE

(* Data type in LON/NetworkVariables *)
TYPE typSnvtTempP : 
STRUCT
	iSnvtTempP : INT;
	bStatusInformation : BYTE; (* bit allocation of bStatusInformation:
	bit 0: NVI update counter LSB
	bit 1: NVI update counter
	bit 2: NVI update counter
	bit 3: NVI update counter MSB
	bit 4: timeout for NVI occurs (MaxRcvTime expired)
	bit 5: reserved
	bit 6: reserved
	bit 7: force NVO update *)
	bInternalUseOnly : BYTE; (* Do not use this byte in your application! *)
END_STRUCT
END_TYPE

(* Data type in LON/NetworkVariables *)
TYPE typSnvtTimeStamp : 
STRUCT
	iYear : INT;
	bMonth : BYTE;
	bDay : BYTE;
	bHour : BYTE;
	bMinute : BYTE;
	bSecond : BYTE;
	bStatusInformation : BYTE; (* bit allocation of bStatusInformation:
	bit 0: NVI update counter LSB
	bit 1: NVI update counter
	bit 2: NVI update counter
	bit 3: NVI update counter MSB
	bit 4: timeout for NVI occurs (MaxRcvTime expired)
	bit 5: reserved
	bit 6: reserved
	bit 7: force NVO update *)
	bInternalUseOnly : BYTE; (* Do not use this byte in your application! *)
END_STRUCT
END_TYPE

(* POU PLC_PRG, ST *)
PROGRAM PLC_PRG
VAR
	Timer1: TON; (* Fast controls tick *)
	Timer2: TON; (* Plant control tick *)
	Timer3: TON; (* Logger timer *)

	T_CIRD01	:	INT;
	T_CIRD02	:	INT;
	T_CIR01		:	INT;
	T_CIR02		:	INT;
	T_ACS		:	INT;
	T_Valve01	:	INT;
	T_Valve02	:	INT;

	SecCircuitLogic	:	BOOL;	(* Secondary circuit request: LOGICAL ON/OFF *)
	SecCircuitReal	:	BOOL;	(* Secondart circuit request: REAL ON/OFF	 *)

	i	:	INT;

	Gain: INT;
	test: BOOL;
	Gain1: REAL;
	Gain2: REAL;
	Gain3: REAL;



	ErroreAcqua: INT;

	StartCAL_Antigelo: RS;
	fAntigelo		:FLT_TAP;  (* Sgnalazione LOG Antigelo  *)

END_VAR
VAR_INPUT RETAIN
	TempStartAnigelo: INT:=30;
	TempStopAnigelo: INT:=50;
	BitAttivazioneAntigelo: WORD;
END_VAR
(******************************************************************************
 ****                           MAIN TASK CODE                             ****
 ******************************************************************************

	Network setup:
		IP  = 192.168.100.2 | MSK = 255.255.255.0
		GW	= 192.168.100.1 | DNS = 192.168.100.1
		SNTP = 193.204.114.232 (3600s) ==> 192.168.100.3

*)

(*==============================*)
(*===== Main status machine ====*)
(*==============================*)
Main_Stm();

(*==============================*)
(*== Running cycle operations ==*)
(*==============================*)
IF SYS.Status>S_INIT_VAR THEN
	(* Execute cycle processes *)
	(* Update LON output variables (needs to be here to obtain only one refresh) *)
	CAL01.Heartbeat( CLIM:=CAL01_Clima );
	(* Execute LON process *)
	Module_1_PRG();

	(* Count water pulses *)
	CTL01(CTL_ST:=CTL01_ST, COUNT:=Ctl01_Counter);
	CTL02(CTL_ST:=CTL02_ST, COUNT:=Ctl02_Counter);
	CTL03(CTL_ST:=CTL03_ST, COUNT:=Ctl03_Counter);

	(* ModBus and CIR *)
	MODB01();

	CIRD02(ModBus:=MODB01, PumpA_AL:=NOT CIRD02_A_AL, PumpB_AL:=NOT CIRD02_B_AL, PumpA_AUTO:=NOT CIRD02_A_AUTO, PumpB_AUTO:=NOT CIRD02_B_AUTO);
	CIRD03(ModBus:=MODB01, PumpA_AL:=NOT CIRD03_A_AL, PumpB_AL:=NOT CIRD03_B_AL, PumpA_AUTO:=NOT CIRD03_A_AUTO, PumpB_AUTO:=NOT CIRD03_B_AUTO,
		   OnOff:=SecCircuitReal);


NodoDaInterrogare:=LIMIT(NodoDaInterrogare,1,5);
IF NodoDaInterrogare>4 THEN NodoDaInterrogare:=1;END_IF;




	(* ModBus TCP and Zigbee sensors *)
	MODB02();

	ZTHL06(ModBus:=MODB02);
	ZTHL07(ModBus:=MODB02);
	ZTHL08(ModBus:=MODB02);
	ZTHL09(ModBus:=MODB02);
	ZTHL10(ModBus:=MODB02);
(*	ZTHL11(ModBus:=MODB02); *)

	(* M-Bus and CTB *)
	MBUS01();

	CTB01(MBUS:=MBUS01);
	CTB02(MBUS:=MBUS01);
END_IF

(*==============================*)
(*== System cycle operations ===*)
(*==============================*)
(* Execute TCP processes *)
Logger_Proc();
Remote_Proc();
(* Update user led *)
USRLED_Update();
(* Execute Cron Editor commands *)
CronEd();

(* Environment temperature *)
IF NOT TPV01.ERR THEN T_AMB := S01;
ELSE T_AMB := Plant_DefaultTAmb;
END_IF


(**** SIMULATION ONLY ****)
(*...*)
END_PROGRAM
ACTION Main_Stm:
CASE Sys.Status OF

	S_STARTUP:
		Sys.Status:=S_INIT_RTC;

	S_INIT_RTC:
		(* Check RTC and update from network *)
		RTC_Update();
		(* Check time *)
		IF Sys.Time_Year>2000 THEN
			Sys.Status:=S_INIT_VAR;
		END_IF

	S_INIT_VAR:
		LogEv(EL_Wrn,EO_SYS,0,1,CONCAT('System_startup_v',WORD_TO_STRING(Plant_SW_VER)));
		Sys.Status:=S_RUNNING;

	S_RUNNING:
		Timer1(IN:=NOT Timer1.Q,PT:=T#50ms);
		IF Timer1.Q THEN
			(* Update meters *)

			(* Update system checks *)
			SYS_Proc();
		END_IF

		Timer2(IN:=NOT Timer2.Q,PT:=T#500ms);
		IF Timer2.Q THEN
			(* Read current date/time *)
			RTC_Update();


			(* Temperature probes *)
			TPV01(IN:=S01);
			TPV02(IN:=S02);
			TPV03(IN:=S03);
			TPV04(IN:=S04);
			TPV05(IN:=S05);
			TPV12(IN:=S12);


			TPV05.Mean();
			T_ACS	:= SEL(TPV05.ERR,TPV05.AVG, 600);


		(* Gestione Ciclo antigelo : in questo impianto il ciclo antigelo è gestito coi crono ambiente *)

			StartCAL_Antigelo(	SET:=(SogliaMinStartAntigelo>TPV03.AVG),
								RESET1:= (TPV03.AVG>SogliaMinStopAntigelo) OR NOT BitAbilitaAntigelo
							);



			fAntigelo(IN:=StartCAL_Antigelo.Q1);
			IF fAntigelo.EVH THEN
				LogEv(EL_Log,EO_SYS,0,11,'Ciclo_Antigelo_Attivato');
			END_IF
			IF fAntigelo.EVL THEN
				LogEv(EL_Log,EO_SYS,0,12,'Ciclo_Antigelo_Disattivato');
			END_IF



			(* Thermostat *)
			THER01(Temperature:=MIN(ZTHL06.OUT_TEMP,ZTHL07.OUT_TEMP));
			CIRD01.OnOff:=SEL(ZTHL06.ERR AND ZTHL07.ERR,THER01.Run,THER01.RunCrono) OR StartCAL_Antigelo.Q1; (* Ala nuova Fan Coil *)


			THER02(Temperature:=MIN(ZTHL08.OUT_TEMP,ZTHL09.OUT_TEMP));
			CIRD02.OnOff:=SEL(ZTHL08.ERR AND ZTHL09.ERR,THER02.Run,THER02.RunCrono) OR StartCAL_Antigelo.Q1; (* Ala vecchia radiatori *)


			THER03(Temperature:=ZTHL10.OUT_TEMP);
			CIR02.OnOff:= SEL(ZTHL10.ERR,THER03.Run,THER03.RunCrono) OR StartCAL_Antigelo.Q1;


		(*	THER04(Temperature:=0, Run=>CIRD03.OnOff);				(*, AntifreezeForce=>CIR01.CIR_RUN_REQ);*) *)

			THER05(Temperature:=T_ACS);
			CIR03.OnOff:=THER05.RunCrono OR StartCAL_Antigelo.Q1;	(* Circolatore *)
			THER06(Temperature:=T_ACS, Run=>CIR01.OnOff);			(* Bollitore *)


			(* CIRs *)
			CIR01(Pump_AL:=NOT CIR01_AL, Pump_ST:=CIR01_ST, Pump_AUTO:=NOT CIR01_AUTO, CIR_EN=>CIR01_EN);
			CIR02(Pump_AL:=NOT CIR02_AL, Pump_ST:=CIR02_ST, Pump_AUTO:=NOT CIR02_AUTO, CIR_EN=>CIR02_EN);
			CIR03(Pump_AL:=NOT CIR03_AL, Pump_ST:=CIR03_ST, Pump_AUTO:=NOT CIR03_AUTO, CIR_EN=>CIR03_EN);

			(* Double CIR (not Modbus) *)
			CIRD01(PumpA_AL:=NOT CIRD01_A_AL, PumpB_AL:=NOT CIRD01_B_AL, PumpA_AUTO:=NOT CIRD01_A_AUTO, PumpB_AUTO:=NOT CIRD01_B_AUTO,
				   PumpA_En=>CIRD01_A_EN, PumpB_En=>CIRD01_B_EN, Tprobe:=T_Valve02);


			(* Calcolo l'errore dell'acqua mandata e ritorno in modo da controllare la velocità delle pompe di mandata *)
			ErroreAcqua:=STRING_TO_INT(CTB01.M1.utFTemp.Value)-STRING_TO_INT(CTB01.M1.utRTemp.Value);

			Gain1:=INT_TO_REAL(PercVelMax-PercVelMin)/INT_TO_REAL(ErroreTempMax-ErroreTempMin);
			Gain2:=Gain1*INT_TO_REAL(ErroreAcqua-ErroreTempMin);
			Gain3:=Gain2 + INT_TO_REAL(PercVelMin);
			Gain:=LIMIT(REAL_TO_INT(Gain3),PercVelMin,PercVelMax);

			CIRD03.VelocitaRichiesta:= Gain;


			(* Secondary circuit heat request *)
			SecCircuitLogic := CIRD01.Ctrl_Run OR CIRD02.Ctrl_Run OR CIR02.Ctrl_Run OR CIR01.Ctrl_Run OR CIR03.Ctrl_Run;
			SecCircuitReal	:= CIRD01.Run OR CIRD01.Run OR CIR02.Run OR CIR01.Run OR CIR03.Run;

			(* Comando Ciroclatore Primario *)
			CIRD03.OnOff := SEL(SecCircuitLogic,FALSE,TRUE) AND SYS.AlarmStop=FALSE;
			CAL01.Run := SEL(SecCircuitLogic,FALSE,CIRD03.Run) AND SYS.AlarmStop=FALSE;


			THER250();			(* Boost *)


			(* Scrivo il setpoint in funzione della curva cliamatica più alta *)

			CAL01.SetPointManuale:=CAL01.Curve_Temp - OffsetSetPointManuale + THER250.SetPoint;
			CAL01.SetPointManuale:=MAX(CAL01.SetPointManuale,SEL(CIR01.OnOff,0,THER06.SetPoint));
			CAL01.SetPointManuale:=MAX(CAL01.SetPointManuale,SEL(VRD01.RUN,0,VRD01.Ctrl_SetPoint));
			CAL01.SetPointManuale:=MAX(CAL01.SetPointManuale,SEL(VRD02.RUN,0,VRD02.Ctrl_SetPoint));
			CAL01(CLIM:=CAL01_Clima,AbilitaSetPointManuale:=TRUE);




			(* Valves *)
			TPV04.Mean();
			T_Valve01 := SEL(TPV04.ERR,TPV04.AVG,Plant_VRD_TDefault);

			VRD01(RUN:=CIRD02.Run,OffsetBoost:=THER250.SetPoint, CLIM:=VRD01_Clima, TEMP:=T_Valve01, STATUS:=VRD01_ST, OUT_CL=>VRD01_CL, OUT_OP=>VRD01_OP);

			TPV12.Mean();
			T_Valve02 := SEL(TPV12.ERR,TPV12.AVG,Plant_VRD_TDefault);

			VRD02(RUN:=CIRD01.Run,OffsetBoost:=THER250.SetPoint, CLIM:=VRD02_Clima, TEMP:=T_Valve02, STATUS:=VRD02_ST, OUT=>VRD02_CTRL);

			(* Check plant status *)

			Lamp( Allarme:=	CAL01.Status_Log=2 OR
 							CTL01.Status_Log=2 OR
							CTL02.Status_Log=2 OR
							CTL03.Status_Log=2 OR
 						  	CIR01.Status_Log=2 OR
  						  	CIR02.Status_Log=2 OR
  						  	CIR03.Status_Log=2 OR
  						  	CIRD01.Status_Log=2 OR
 						  	CIRD02.Status_Log=2 OR
						  	CIRD03.Status_Log=2 OR
							TPV01.Status_Log=2 OR
							TPV02.Status_Log=2 OR
							TPV03.Status_Log=2 OR
							TPV04.Status_Log=2 OR
							TPV05.Status_Log=2 OR
							TPV12.Status_Log=2 OR
							THER01.Status_Log=2 OR
							THER02.Status_Log=2 OR
							THER03.Status_Log=2 OR
							THER04.Status_Log=2 OR
							THER05.Status_Log=2 OR
							THER06.Status_Log=2 OR
							THER250.Status_Log=2 OR
							VRD01.Status_Log=2 OR
							VRD02.Status_Log=2 OR
							CTB01.Status_Log=2 OR
							CTB02.Status_Log=2 OR
							MODB01.Status_Log=2 OR
							MODB02.Status_Log=2 OR
							MBUS01.Status_Log=2 OR
							ZTHL07.Status_Log=2 OR
							ZTHL08.Status_Log=2 OR
							ZTHL09.Status_Log=2 OR
							ZTHL10.Status_Log=2	,
							Warning:=CAL01.Status_Log=1 OR
 							CTL01.Status_Log=1 OR
							CTL02.Status_Log=1 OR
							CTL03.Status_Log=1 OR
 						  	CIR01.Status_Log=1 OR
  						  	CIR02.Status_Log=1 OR
  						  	CIR03.Status_Log=1 OR
  						  	CIRD01.Status_Log=1 OR
 						  	CIRD02.Status_Log=1 OR
						  	CIRD03.Status_Log=1 OR
							TPV01.Status_Log=1 OR
							TPV02.Status_Log=1 OR
							TPV03.Status_Log=1 OR
							TPV04.Status_Log=1 OR
							TPV05.Status_Log=1 OR
							TPV12.Status_Log=1 OR
							THER01.Status_Log=1 OR
							THER02.Status_Log=1 OR
							THER03.Status_Log=1 OR
							THER04.Status_Log=1 OR
							THER05.Status_Log=1 OR
							THER06.Status_Log=1 OR
							THER250.Status_Log=1 OR
							VRD01.Status_Log=1 OR
							VRD02.Status_Log=1 OR
							CTB01.Status_Log=1 OR
							CTB02.Status_Log=1 OR
							MODB01.Status_Log=1 OR
							MODB02.Status_Log=1 OR
							MBUS01.Status_Log=1 OR
							ZTHL07.Status_Log=1 OR
							ZTHL08.Status_Log=1 OR
							ZTHL09.Status_Log=1 OR
							ZTHL10.Status_Log=1	,
							AllarmeLampada=>LAMP_AL
							);




			(* Test toggle *)
			(*IF TEST1 THEN TEST1:=FALSE; ELSE TEST1:=TRUE; END_IF*)
		END_IF

		Timer3(IN:=NOT Timer3.Q,PT:=T#5m);
		IF Timer3.Q THEN
			(* Trig logger *)
			LogTrig();
			(* Execute temporary CSV logger *)
			(*CSV_Log();*)
		END_IF

	S_SHUTDOWN:
		(* Stop sistema *)
		Sys.Status:=S_STARTUP;

	S_HALT:
		(* Aspetta uscita manuale *)
		Sys.Status:=S_STARTUP;

ELSE
	Sys.Status:=S_STARTUP;
END_CASE;
END_ACTION

(* POU Utils Functions/FLT_TAP, ST *)
FUNCTION_BLOCK FLT_TAP
VAR_INPUT
	IN		: BOOL;
	TAP		: BYTE:=4;
	INITEV	: BOOL:=TRUE;
END_VAR
VAR_OUTPUT
	OUT		: BOOL;
	EVH		: BOOL;
	EVL		: BOOL;
END_VAR
VAR
	init	: BOOL:=FALSE;
	cnt		: BYTE;
END_VAR
EVH:=FALSE;
EVL:=FALSE;

IF NOT init THEN
	init := TRUE;
	IF INITEV THEN
		OUT  := NOT IN;
		cnt  := TAP;
	ELSE
		OUT  := IN;
	END_IF
END_IF

IF OUT<>IN THEN
	cnt:=cnt+1;
	IF cnt>TAP THEN
		OUT:=IN;
		cnt:=0;
		IF OUT THEN EVH:=TRUE; ELSE EVL:=TRUE; END_IF
	END_IF
ELSE
	cnt:=0;
END_IF
END_FUNCTION_BLOCK

(* POU LON/Module_1/Module_1_PRG, FBD *)
PROGRAM Module_1_PRG
VAR
	(* Automatic added code, do not change! *)
	LonMaster : Module_1_LonMaster;
	SFPTnodeObject : Module_1_SFPTnodeObject;
	Virtualfunctionalblock : Module_1_Virtualfunctionalblock;

	InData_LON AT %IB0 : ARRAY[0..23] OF BYTE;
	OutData_LON AT %QB0 : ARRAY[0..23] OF BYTE;
	(***** End of automatic added code. *****)

	(* Add your code here. *)
	LonState: BOOL;
	LonReset: BOOL;

END_VAR
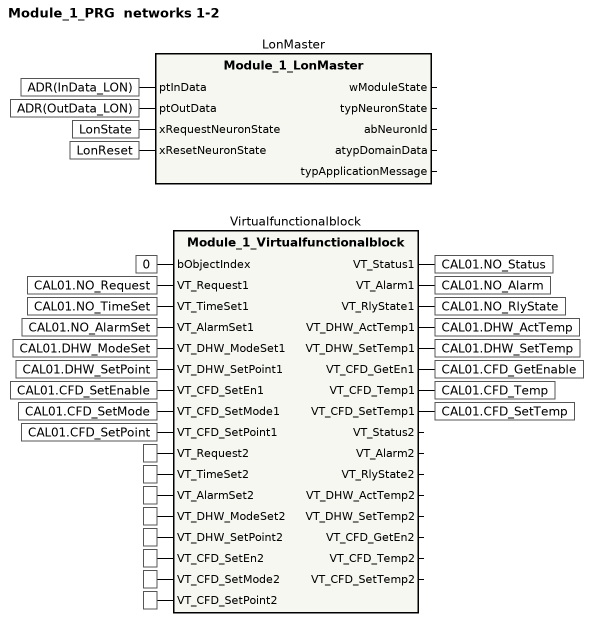
_FBD_ (* Function Block Diagram *)
NETWORK 1 (* Added by code generator *)
	LonMaster:Module_1_LonMaster(ptInData: ADR(InData_LON), ptOutData: ADR(OutData_LON), xRequestNeuronState: LonState, xResetNeuronState: LonReset)
NETWORK 2
	Virtualfunctionalblock:Module_1_Virtualfunctionalblock(bObjectIndex: 0, VT_Request1: CAL01.NO_Request, VT_TimeSet1: CAL01.NO_TimeSet, VT_AlarmSet1: CAL01.NO_AlarmSet, VT_DHW_ModeSet1: CAL01.DHW_ModeSet, VT_DHW_SetPoint1: CAL01.DHW_SetPoint, VT_CFD_SetEn1: CAL01.CFD_SetEnable, VT_CFD_SetMode1: CAL01.CFD_SetMode, VT_CFD_SetPoint1: CAL01.CFD_SetPoint, VT_Request2: , VT_TimeSet2: , VT_AlarmSet2: , VT_DHW_ModeSet2: , VT_DHW_SetPoint2: , VT_CFD_SetEn2: , VT_CFD_SetMode2: , VT_CFD_SetPoint2: , VT_Alarm1 => CAL01.NO_Alarm, VT_RlyState1 => CAL01.NO_RlyState, VT_DHW_ActTemp1 => CAL01.DHW_ActTemp, VT_DHW_SetTemp1 => CAL01.DHW_SetTemp, VT_CFD_GetEn1 => CAL01.CFD_GetEnable, VT_CFD_Temp1 => CAL01.CFD_Temp, VT_CFD_SetTemp1 => CAL01.CFD_SetTemp) => CAL01.NO_Status
_END_FBD_
(* the same logic as Structured Text *)
(* Network 1 *)
LonMaster(ptInData := ADR(InData_LON), ptOutData := ADR(OutData_LON), xRequestNeuronState := LonState, xResetNeuronState := LonReset);
(* Network 2: see the listing above *)
END_PROGRAM

(* POU LON/Module_1/Master/Module_1_LonMaster, ST *)
FUNCTION_BLOCK Module_1_LonMaster
(******************************************)
(* Automatic generated code, do not edit! *)
(******************************************)
VAR_INPUT
	ptInData  : POINTER TO BYTE;
	ptOutData : POINTER TO BYTE;
	xRequestNeuronState : BOOL;
	xResetNeuronState : BOOL;
END_VAR
VAR_OUTPUT
	wModuleState : WORD; (* bit coded wModuleState:
	15: communication to I/O-module interrupted (error)
	14 - 08: reserved
	07: ready for Neuron initialization
	06: Neuron active
	05: user interface active
	04: internal module communication interrupted (error)
	03: CP synchronization running
	02: Neuron is configured online
	01 - 00: reserved *)

	typNeuronState : NeuronState;
	abNeuronId : ARRAY[0..5] OF BYTE;
	atypDomainData : ARRAY[0..1] OF DomainData;
	typApplicationMessage : ApplicationMessageData;
END_VAR
VAR
	bInternalCode : BYTE;
	bNvIndex : BYTE;
	wCpIndex : WORD;
	lonCom : FbLonBasicCommunication;

	xInitIsStarted : BOOL := FALSE;

	TimeoutTimer : TON;
	timeOutTime : TIME := T#1000ms;
	xStateMachineIsChecked : BOOL;
	xTimerStart : BOOL;

	iDomainTable : INT;
	xSendRequestPending : BOOL;
	trigRequest : R_TRIG;
	trigReset : R_TRIG;

	abMbxRxPrio0Buf: ARRAY [0..309] OF BYTE;
	abMbxRxPrio1Buf: ARRAY [0..517] OF BYTE;
	aMbxRxBufSize: ARRAY [0..1] OF UINT := 310, 518;
	aMbxRxBufList: ARRAY [0..1] OF POINTER TO BYTE;
	afbMbxRxFb: ARRAY [0..1] OF MBX2_RX_DEFRAG;
	astMbxRxCtx: ARRAY [0..1] OF stMbx2DefragContext;

	abMbxTxPrio0Buf: ARRAY [0..309] OF BYTE;
	abMbxTxPrio1Buf: ARRAY [0..517] OF BYTE;
	aMbxTxBufSize: ARRAY [0..1] OF UINT := 310, 518;
	aMbxTxBufList: ARRAY [0..1] OF POINTER TO BYTE;
	afbMbxTxFb: ARRAY [0..1] OF MBX2_TX_FRAG;

	astMbxTrackContext: ARRAY [0..0] OF stMbx2TrackContext;
END_VAR
VAR CONSTANT
END_VAR
aMbxRxBufList[0] := ADR(abMbxRxPrio0Buf[0]);
aMbxRxBufList[1] := ADR(abMbxRxPrio1Buf[0]);

aMbxTxBufList[0] := ADR(abMbxTxPrio0Buf[0]);
aMbxTxBufList[1] := ADR(abMbxTxPrio1Buf[0]);

mbxModule_1.Ressources.pDefragBufList := ADR(aMbxRxBufList);
mbxModule_1.Ressources.pDefragBufSizeList := ADR(aMbxRxBufSize);
mbxModule_1.Ressources.pDefragCtxPtrList := ADR(astMbxRxCtx);
mbxModule_1.Ressources.pDefragFbList := ADR(afbMbxRxFb);
mbxModule_1.Ressources.pFragBufList := ADR(aMbxTxBufList);
mbxModule_1.Ressources.pFragBufSizeList := ADR(aMbxTxBufSize);
mbxModule_1.Ressources.pFragFbList := ADR(afbMbxTxFb);

mbxModule_1.Ressources.unMaxAvailableRxPrioIndex := 1;
mbxModule_1.Ressources.unMaxAvailableTxPrioIndex := 1;

mbxModule_1.Ressources.pTrackStList := ADR(astMbxTrackContext);
mbxModule_1.Ressources.unMaxAvailableTrackIndex := 0;

mbxModule_1.Ressources.pabRxWin := ptInData + 1;
mbxModule_1.Ressources.pabTxWin := ptOutData + 1;
mbxModule_1.Ressources.bTxWinSize := 23;
mbxModule_1.Ressources.bRxWinSize := 23;

IF (mbxModule_1.bStatus.2 = TRUE) OR (mbxModule_1.bStatus.1 = TRUE) THEN
	mbxModule_1.MBX_RESET();
	xInitRunning_Module_1 := TRUE;
	xInitIsStarted := FALSE;
END_IF
mbxModule_1.MBX_CYCLE();

IF (mbxModule_1.bStatus.0 <> TRUE) THEN 
	wModuleState := 16#8000;
	RETURN;
ELSE
	wModuleState.15 := FALSE;
END_IF

xStateMachineIsChecked := FALSE;
IF xInitRunning_Module_1 = TRUE THEN
	IF xInitIsStarted = FALSE THEN
		SetParameter();
		lonCom.eInitState := INIT_SND_SGNTR_REQ;
		lonCom.CheckInitState();
		xInitIsStarted := TRUE;
		xStateMachineIsChecked := TRUE;
	END_IF
END_IF

typApplicationMessage.xMsgRcvd := FALSE;
typApplicationMessage.xRspRcvd := FALSE;
ResetNviUpdate();
WHILE (mbxModule_1.xRxPending) DO
	unLastLen_mbxModule_1 := mbxModule_1.unRxLen;
	mbxModule_1.pbRxData := ADR(InDataTelegram_Module_1);
	mbxModule_1.MBX_RETRIEVE();
	IF (mbxModule_1.nError <> MBX_OK) THEN EXIT; END_IF;
	bInternalCode := InDataTelegram_Module_1[0];

	IF (xInitRunning_Module_1 = TRUE) AND (lonCom.eInitState <> INIT_TRANSFER_CFG) THEN
		IF (FuCheckForValidInitCode(bInternalCode)) THEN
			SetParameter();
			lonCom.unLastLen := unLastLen_mbxModule_1;
			lonCom.CheckInitState();
			xInitRunning_Module_1 := NOT lonCom.xInitDone;
			xStateMachineIsChecked := TRUE;
		END_IF
	END_IF

	IF (bInternalCode = M2C_NVI_UPDT_OCCD) OR (bInternalCode = M2C_NV_VALUE_RSP) OR (bInternalCode = M2C_NVI_UPDT_TOUT) THEN
		bNvIndex := InDataTelegram_Module_1[1];
		CASE bNvIndex OF
			0, 2, 4: Module_1_PRG.SFPTnodeObject.DataReceived();
			6, 8, 10, 12, 14, 16, 18, 20, 22, 24, 26, 28, 30, 32, 34, 36: Module_1_PRG.Virtualfunctionalblock.DataReceived();

		END_CASE;
	ELSIF (bInternalCode = M2C_CP_VALUE_RSP) THEN
		wCpIndex := InDataTelegram_Module_1[1] OR (InDataTelegram_Module_1[2] * 256);
		CASE wCpIndex OF

		END_CASE;
	ELSIF (bInternalCode = M2C_LON_MSG_RCVD) OR (bInternalCode = M2C_LON_RSP_RCVD) THEN
		ApplMsgReceived();
	ELSIF (bInternalCode = M2C_STATUS_RSP) THEN
		wModuleState := (wModuleState AND 16#FF00) + InDataTelegram_Module_1[1];
	ELSIF (bInternalCode = M2C_NEURON_ID) THEN
		FuMemCopy(ADR(InDataTelegram_Module_1[1]), ADR(abNeuronId), 6);
	ELSIF (bInternalCode = M2C_DOMAIN_DATA) THEN
		DomainDataRcvd();
	ELSIF (bInternalCode = M2C_MICRO_SERVER_STATUS_RSP) THEN
		NeuronStateRcvd();
	END_IF
END_WHILE

IF (xInitRunning_Module_1 = TRUE) AND ((lonCom.xCallStateMachine = TRUE) OR (TimeoutTimer.Q = TRUE)) AND (NOT xStateMachineIsChecked) THEN
	SetParameter();
	lonCom.xTimeOut := TimeoutTimer.Q;
	lonCom.CheckInitState();
END_IF
TimeoutTimer(IN:=lonCom.xTimerStart, PT:=timeOutTime);

trigRequest(CLK := xRequestNeuronState);
trigReset(CLK := xResetNeuronState);
IF (trigRequest.Q OR trigReset.Q) THEN
	RequestNeuronState();
END_IF
END_FUNCTION_BLOCK
ACTION ApplMsgReceived:
IF (InDataTelegram_Module_1[0] = M2C_LON_MSG_RCVD) THEN
	typApplicationMessage.typService := InDataTelegram_Module_1[1] AND 16#30;
	typApplicationMessage.bSourceSubnetId := InDataTelegram_Module_1[2];
	typApplicationMessage.bSourceNodeId := InDataTelegram_Module_1[3];
	typApplicationMessage.bCorrelator := InDataTelegram_Module_1[4];
	typApplicationMessage.bCode :=  InDataTelegram_Module_1[5];
	typApplicationMessage.bDataLength := UINT_TO_BYTE(unLastLen_mbxModule_1 - 6);
	IF typApplicationMessage.bDataLength > 48 THEN typApplicationMessage.bDataLength := 48; END_IF;
	FuMemSet(ADR(typApplicationMessage.abData), 0, SIZEOF(typApplicationMessage.abData));
	IF typApplicationMessage.bDataLength > 0 THEN
		FuMemCopy(ADR(InDataTelegram_Module_1[6]), ADR(typApplicationMessage.abData), typApplicationMessage.bDataLength);
	END_IF
	typApplicationMessage.xMsgRcvd := TRUE;
ELSE
	typApplicationMessage.typService := LON_RESPONSE;
	typApplicationMessage.bSourceSubnetId := InDataTelegram_Module_1[1];
	typApplicationMessage.bSourceNodeId := InDataTelegram_Module_1[2];
	typApplicationMessage.bCorrelator := 0;
	typApplicationMessage.bCode :=  InDataTelegram_Module_1[3];
	typApplicationMessage.bDataLength := UINT_TO_BYTE(unLastLen_mbxModule_1 - 4);
	IF typApplicationMessage.bDataLength > 48 THEN typApplicationMessage.bDataLength := 48; END_IF;
	FuMemSet(ADR(typApplicationMessage.abData), 0, SIZEOF(typApplicationMessage.abData));
	IF typApplicationMessage.bDataLength > 0 THEN
		FuMemCopy(ADR(InDataTelegram_Module_1[4]), ADR(typApplicationMessage.abData), typApplicationMessage.bDataLength);
	END_IF
	typApplicationMessage.xRspRcvd := TRUE;
END_IF
END_ACTION
ACTION DomainDataRcvd:
IF (unLastLen_mbxModule_1 = 17) THEN
	iDomainTable := InDataTelegram_Module_1[1];
	IF (iDomainTable < 0) OR (iDomainTable > 1) THEN RETURN; END_IF
	FuMemCopy(ADR(InDataTelegram_Module_1[2]), ADR(atypDomainData[iDomainTable].abDomainId), 6);
	atypDomainData[iDomainTable].bSubnet := InDataTelegram_Module_1[8];
	atypDomainData[iDomainTable].xIsNonClone := InDataTelegram_Module_1[9].7;
	atypDomainData[iDomainTable].bNodeId := InDataTelegram_Module_1[9] AND 16#7F;
	atypDomainData[iDomainTable].xIsInvalid := InDataTelegram_Module_1[10].7;
	atypDomainData[iDomainTable].bDomainIdLength := InDataTelegram_Module_1[10] AND 16#7F;
	FuMemCopy(ADR(InDataTelegram_Module_1[11]), ADR(atypDomainData[iDomainTable].abAuthenticationKey), 6);
END_IF
END_ACTION
ACTION NeuronStateRcvd:
IF (unLastLen_mbxModule_1 = 16) THEN
	typNeuronState.wCrcError := InDataTelegram_Module_1[1] + InDataTelegram_Module_1[2] * 256;
	typNeuronState.wTransactionTimeouts := InDataTelegram_Module_1[3] + InDataTelegram_Module_1[4] * 256;
	typNeuronState.wReceiveTransactionBuffersFull := InDataTelegram_Module_1[5] + InDataTelegram_Module_1[6] * 256;
	typNeuronState.wLostMessages := InDataTelegram_Module_1[7] + InDataTelegram_Module_1[8] * 256;
	typNeuronState.wMissedMessages := InDataTelegram_Module_1[9] + InDataTelegram_Module_1[10] * 256;
	typNeuronState.bResetCause := InDataTelegram_Module_1[11];
	typNeuronState.bNodeState := InDataTelegram_Module_1[12];
	typNeuronState.bFirmwareVersion := InDataTelegram_Module_1[13];
	typNeuronState.bLastErrorLogged := InDataTelegram_Module_1[14];
	typNeuronState.bModelNumber := InDataTelegram_Module_1[15];
END_IF
END_ACTION
ACTION RequestNeuronState:
OutDataTelegram_Module_1[0] := C2M_MICRO_SERVER_STATUS_QRY;
OutDataTelegram_Module_1[1] := BOOL_TO_BYTE(trigReset.Q);

mbxModule_1.bTxPrio := 1;
mbxModule_1.bTxProtID := 0;
mbxModule_1.pbTxData := ADR(OutDataTelegram_Module_1);
mbxModule_1.unTxLen := 2;
mbxModule_1.MBX_SEND();

IF (mbxModule_1.nError <> MBX_OK) THEN
	RETURN;
END_IF
END_ACTION
ACTION ResetNviUpdate:
Module_1_PRG.SFPTnodeObject.ResetNviUpdate();
Module_1_PRG.Virtualfunctionalblock.ResetNviUpdate();
END_ACTION
ACTION SetParameter:
lonCom.pMbx 			:= ADR(mbxModule_1);
lonCom.pInData 			:= ADR(InDataTelegram_Module_1);
lonCom.pOutData 		:= ADR(OutDataTelegram_Module_1);
lonCom.pTimer			:= ADR(TimeoutTimer);

lonCom.pActualSignature	:= ADR(abSignature_Module_1);
lonCom.pConfigBlock := ADR(abInterface_Module_1);
lonCom.wConfigSize 		:= wConfigSize_Module_1;
END_ACTION

(* POU LON/Module_1/NV_Interface/Module_1_SFPTnodeObject, ST *)
FUNCTION_BLOCK Module_1_SFPTnodeObject
(******************************************)
(* Automatic generated code, do not edit! *)
(******************************************)
VAR_INPUT
	bObjectIndex : BYTE := 0;
	nvoStatus : typSnvtObjStatus;
	nvoFileStat : typSnvtFileStatus;

END_VAR
VAR_OUTPUT
	nviRequest : typSnvtObjRequest;
	nviFileReq : typSnvtFileReq;
	nviFilePos : typSnvtFilePos;

END_VAR
VAR
	xSetOnce : BOOL := TRUE;
	xDataInUpdated : BOOL := FALSE;
	nvoStatusLast: typSnvtObjStatus;
	nvoFileStatLast: typSnvtFileStatus;

	cmd : BYTE;
	z : INT;
	bNvRelativeIdx : BYTE;
	bNvAbsoluteIdx : BYTE;
	wCpRelativeIdx : WORD;
	wCpAbsoluteIdx : WORD;
END_VAR
VAR CONSTANT
	bNvStartIndex : BYTE := 0;
	wCpStartIndex : WORD := 65535;
	bLmoCount : BYTE := 1;
END_VAR
IF (xInitRunning_Module_1 = TRUE) AND (xSetOnce = TRUE) THEN
	xSetOnce := FALSE;
	CachePointers();
	SetUpdateFlags();
END_IF

CheckUpdateFlags();
IF (xInitRunning_Module_1 = FALSE) AND (xDataInUpdated = FALSE) THEN
	IF (mbxModule_1.bStatus.0) THEN
		SendValueRequest();
	END_IF
END_IF

IF (xInitRunning_Module_1 = FALSE) AND (mbxModule_1.bStatus.0) THEN
	xSetOnce := TRUE;
	xDataInUpdated := FALSE;
	IF ((NOT FuMemCompare(ADR(nvoStatusLast), ADR(nvoStatus), ADR(nvoStatus.bStatusInformation) - ADR(nvoStatus))) OR (nvoStatus.bStatusInformation.7 = TRUE) OR (nvoStatusLast.bInternalUseOnly.1 = TRUE)) THEN
		FuSnvtObjStatusToRaw(ADR(nvoStatus), ADR(OutDataTelegram_Module_1[2]));

		bNvAbsoluteIdx := bNvStartIndex + bObjectIndex + (1 * bLmoCount);

		IF (FuDoNvoUpdate_Module_1(ADR(nvoStatus), ADR(nvoStatusLast), ADR(nvoStatus.bInternalUseOnly), ADR(nvoStatusLast.bInternalUseOnly), ADR(nvoStatus.bStatusInformation), bNvAbsoluteIdx, 6, SIZEOF(nvoStatus)) = FALSE) THEN
			RETURN;
		END_IF
	END_IF
	IF ((NOT FuMemCompare(ADR(nvoFileStatLast), ADR(nvoFileStat), ADR(nvoFileStat.bStatusInformation) - ADR(nvoFileStat))) OR (nvoFileStat.bStatusInformation.7 = TRUE) OR (nvoFileStatLast.bInternalUseOnly.1 = TRUE)) THEN
		FuSnvtFileStatusToRaw(ADR(nvoFileStat), ADR(OutDataTelegram_Module_1[2]));

		bNvAbsoluteIdx := bNvStartIndex + bObjectIndex + (3 * bLmoCount);

		IF (FuDoNvoUpdate_Module_1(ADR(nvoFileStat), ADR(nvoFileStatLast), ADR(nvoFileStat.bInternalUseOnly), ADR(nvoFileStatLast.bInternalUseOnly), ADR(nvoFileStat.bStatusInformation), bNvAbsoluteIdx, 27, SIZEOF(nvoFileStat)) = FALSE) THEN
			RETURN;
		END_IF
	END_IF

END_IF
END_FUNCTION_BLOCK
ACTION CachePointers:
;
END_ACTION
ACTION CheckUpdateFlags:
xDataInUpdated := (NOT nviRequest.bInternalUseOnly.0) AND (NOT nviFileReq.bInternalUseOnly.0) AND (NOT nviFilePos.bInternalUseOnly.0) AND TRUE;
END_ACTION
ACTION DataReceived:
cmd := InDataTelegram_Module_1[0];
IF (cmd = M2C_NVI_UPDT_OCCD) OR (cmd = M2C_NV_VALUE_RSP) OR (cmd = M2C_NVI_UPDT_TOUT) THEN
	bNvRelativeIdx := (InDataTelegram_Module_1[1] - bNvStartIndex - bObjectIndex) / bLmoCount;
	CASE bNvRelativeIdx OF
	0:
		IF (cmd = M2C_NVI_UPDT_OCCD) OR (cmd = M2C_NV_VALUE_RSP) THEN
			IF (unLastLen_mbxModule_1 = (2 + 3)) THEN
				FuRawToSnvtObjRequest(ADR(InDataTelegram_Module_1[2]), ADR(nviRequest));
				nviRequest.bInternalUseOnly.0 := FALSE;
				nviRequest.bStatusInformation := FuInkrementNviStatus(nviRequest.bStatusInformation);
			ELSIF (unLastLen_mbxModule_1 = 2) THEN
				nviRequest.bStatusInformation := FuInkrementNviStatus(nviRequest.bStatusInformation);
			END_IF
		ELSIF (cmd = M2C_NVI_UPDT_TOUT) THEN
			IF (unLastLen_mbxModule_1 = 3) THEN
				nviRequest.bStatusInformation.4 := BYTE_TO_BOOL(InDataTelegram_Module_1[2]);
			END_IF
		END_IF
	2:
		IF (cmd = M2C_NVI_UPDT_OCCD) OR (cmd = M2C_NV_VALUE_RSP) THEN
			IF (unLastLen_mbxModule_1 = (2 + 12)) THEN
				FuRawToSnvtFileReq(ADR(InDataTelegram_Module_1[2]), ADR(nviFileReq));
				nviFileReq.bInternalUseOnly.0 := FALSE;
				nviFileReq.bStatusInformation := FuInkrementNviStatus(nviFileReq.bStatusInformation);
			ELSIF (unLastLen_mbxModule_1 = 2) THEN
				nviFileReq.bStatusInformation := FuInkrementNviStatus(nviFileReq.bStatusInformation);
			END_IF
		ELSIF (cmd = M2C_NVI_UPDT_TOUT) THEN
			IF (unLastLen_mbxModule_1 = 3) THEN
				nviFileReq.bStatusInformation.4 := BYTE_TO_BOOL(InDataTelegram_Module_1[2]);
			END_IF
		END_IF
	4:
		IF (cmd = M2C_NVI_UPDT_OCCD) OR (cmd = M2C_NV_VALUE_RSP) THEN
			IF (unLastLen_mbxModule_1 = (2 + 6)) THEN
				FuRawToSnvtFilePos(ADR(InDataTelegram_Module_1[2]), ADR(nviFilePos));
				nviFilePos.bInternalUseOnly.0 := FALSE;
				nviFilePos.bStatusInformation := FuInkrementNviStatus(nviFilePos.bStatusInformation);
			ELSIF (unLastLen_mbxModule_1 = 2) THEN
				nviFilePos.bStatusInformation := FuInkrementNviStatus(nviFilePos.bStatusInformation);
			END_IF
		ELSIF (cmd = M2C_NVI_UPDT_TOUT) THEN
			IF (unLastLen_mbxModule_1 = 3) THEN
				nviFilePos.bStatusInformation.4 := BYTE_TO_BOOL(InDataTelegram_Module_1[2]);
			END_IF
		END_IF

	END_CASE
ELSIF (cmd = M2C_CP_VALUE_RSP) THEN
	wCpRelativeIdx := ((InDataTelegram_Module_1[1] + InDataTelegram_Module_1[2] * 256) - wCpStartIndex - bObjectIndex) / bLmoCount;
	CASE wCpRelativeIdx OF

	END_CASE
END_IF
END_ACTION
ACTION ResetNviUpdate:
nviRequest.bStatusInformation := nviRequest.bStatusInformation AND 16#F8;
nviFileReq.bStatusInformation := nviFileReq.bStatusInformation AND 16#F8;
nviFilePos.bStatusInformation := nviFilePos.bStatusInformation AND 16#F8;
;
END_ACTION
ACTION SendValueRequest:
IF (FuSendNviValueReq_Module_1(ADR(nviRequest.bInternalUseOnly), bNvStartIndex + bObjectIndex + (0 * bLmoCount)) = FALSE) THEN
	RETURN;
END_IF

IF (FuSendNviValueReq_Module_1(ADR(nviFileReq.bInternalUseOnly), bNvStartIndex + bObjectIndex + (2 * bLmoCount)) = FALSE) THEN
	RETURN;
END_IF

IF (FuSendNviValueReq_Module_1(ADR(nviFilePos.bInternalUseOnly), bNvStartIndex + bObjectIndex + (4 * bLmoCount)) = FALSE) THEN
	RETURN;
END_IF

;
END_ACTION
ACTION SetUpdateFlags:
nviRequest.bInternaluseOnly.0 := TRUE;
nvoStatusLast.bInternaluseOnly.1 := TRUE;
nvoStatusLast.bInternaluseOnly.7 := FALSE;
nviFileReq.bInternaluseOnly.0 := TRUE;
nvoFileStatLast.bInternaluseOnly.1 := TRUE;
nvoFileStatLast.bInternaluseOnly.7 := FALSE;
nviFilePos.bInternaluseOnly.0 := TRUE;
;
END_ACTION

(* POU LON/Shared/Internal/FuSnvtObjStatusToRaw, ST *)
FUNCTION FuSnvtObjStatusToRaw : BOOL
(******************************************)
(* Automatic generated code, do not edit! *)
(******************************************)
VAR_INPUT
	NvDataIn :  POINTER TO typSnvtObjStatus;
	DataOut : POINTER TO ARRAY[0..5] OF BYTE;
END_VAR
VAR
END_VAR
DataOut^[0] := WORD_TO_BYTE(SHR(NvDataIn^.wObjectId, 8));
DataOut^[1] := WORD_TO_BYTE(NvDataIn^.wObjectId);

DataOut^[2] := NvDataIn^.bBitfieldByteOffset2;

DataOut^[3] := NvDataIn^.bBitfieldByteOffset3;

DataOut^[4] := NvDataIn^.bBitfieldByteOffset4;

DataOut^[5] := NvDataIn^.bBitfieldByteOffset5;

FuSnvtObjStatusToRaw := TRUE;
END_FUNCTION

(* POU LON/Module_1/Internal/FuDoNvoUpdate_Module_1, ST *)
FUNCTION FuDoNvoUpdate_Module_1 : BOOL
(******************************************)
(* Automatic generated code, do not edit! *)
(******************************************)
VAR_INPUT
	ptNvo : POINTER TO BYTE;
	ptNvoLast : POINTER TO BYTE;
	ptNvoInternalUse : POINTER TO BYTE;
	ptNvoLastInternalUse : POINTER TO BYTE;
	ptNvoStatusInformation : POINTER TO BYTE;
	bNvoIndex : BYTE;
	uiNvoLength : UINT;
	uiNvoVariableLength : UINT;
END_VAR
IF (ptNvoLastInternalUse^.1 = TRUE) AND (ptNvoStatusInformation^.7 = FALSE) THEN
	OutDataTelegram_Module_1[0] := C2M_NV_VALUE;
ELSE
	OutDataTelegram_Module_1[0] := C2M_NVO_PROPAGATE;
END_IF
OutDataTelegram_Module_1[1] := bNvoIndex;

mbxModule_1.bTxPrio := BOOL_TO_BYTE(ptNvoLastInternalUse^.7);
mbxModule_1.bTxProtID := 0;
mbxModule_1.pbTxData := ADR(OutDataTelegram_Module_1);
mbxModule_1.unTxLen := 2 + uiNvoLength;
mbxModule_1.MBX_SEND();

IF (mbxModule_1.nError <> MBX_OK) THEN
	FuDoNvoUpdate_Module_1 := FALSE;
	RETURN;
END_IF

ptNvoLastInternalUse^.1 := FALSE;
ptNvoInternalUse^ := ptNvoLastInternalUse^;
FuMemCopy(ptNvo, ptNvoLast, uiNvoVariableLength);

FuDoNvoUpdate_Module_1 := TRUE;
END_FUNCTION

(* POU LON/Shared/Internal/FuSnvtFileStatusToRaw, ST *)
FUNCTION FuSnvtFileStatusToRaw : BOOL
(******************************************)
(* Automatic generated code, do not edit! *)
(******************************************)
VAR_INPUT
	NvDataIn :  POINTER TO typSnvtFileStatus;
	DataOut : POINTER TO ARRAY[0..26] OF BYTE;
END_VAR
VAR
END_VAR
DataOut^[0] := NvDataIn^.bStatus;

DataOut^[1] := WORD_TO_BYTE(SHR(NvDataIn^.wNumberOfFiles, 8));
DataOut^[2] := WORD_TO_BYTE(NvDataIn^.wNumberOfFiles);

DataOut^[3] := WORD_TO_BYTE(SHR(NvDataIn^.wSelectedFile, 8));
DataOut^[4] := WORD_TO_BYTE(NvDataIn^.wSelectedFile);

DataOut^[5] := NvDataIn^.abAdr[0];
DataOut^[6] := NvDataIn^.abAdr[1];
DataOut^[7] := NvDataIn^.abAdr[2];
DataOut^[8] := NvDataIn^.abAdr[3];
DataOut^[9] := NvDataIn^.abAdr[4];
DataOut^[10] := NvDataIn^.abAdr[5];
DataOut^[11] := NvDataIn^.abAdr[6];
DataOut^[12] := NvDataIn^.abAdr[7];
DataOut^[13] := NvDataIn^.abAdr[8];
DataOut^[14] := NvDataIn^.abAdr[9];
DataOut^[15] := NvDataIn^.abAdr[10];
DataOut^[16] := NvDataIn^.abAdr[11];
DataOut^[17] := NvDataIn^.abAdr[12];
DataOut^[18] := NvDataIn^.abAdr[13];
DataOut^[19] := NvDataIn^.abAdr[14];
DataOut^[20] := NvDataIn^.abAdr[15];
DataOut^[21] := NvDataIn^.abAdr[16];
DataOut^[22] := NvDataIn^.abAdr[17];
DataOut^[23] := NvDataIn^.abAdr[18];
DataOut^[24] := NvDataIn^.abAdr[19];
DataOut^[25] := NvDataIn^.abAdr[20];
DataOut^[26] := NvDataIn^.abAdr[21];

FuSnvtFileStatusToRaw := TRUE;
END_FUNCTION

(* POU LON/Module_1/Internal/FuSendNviValueReq_Module_1, ST *)
FUNCTION FuSendNviValueReq_Module_1 : BOOL
(******************************************)
(* Automatic generated code, do not edit! *)
(******************************************)
VAR_INPUT
	ptInternalUseOnly : POINTER TO BYTE;
	bNvIndex : BYTE;
END_VAR
IF ptInternalUseOnly^.0 = TRUE THEN
	OutDataTelegram_Module_1[0] := C2M_NV_VALUE_QRY;
	OutDataTelegram_Module_1[1] := bNvIndex;

	mbxModule_1.bTxPrio := 1;
	mbxModule_1.bTxProtID := 0;
	mbxModule_1.pbTxData := ADR(OutDataTelegram_Module_1);
	mbxModule_1.unTxLen := 2;
	mbxModule_1.MBX_SEND();

	IF (mbxModule_1.nError <> MBX_OK) THEN
		FuSendNviValueReq_Module_1 := FALSE;
		RETURN;
	END_IF
	ptInternalUseOnly^.0 := FALSE;
END_IF

FuSendNviValueReq_Module_1 := TRUE;
END_FUNCTION

(* POU LON/Module_1/NV_Interface/Module_1_Virtualfunctionalblock, ST *)
FUNCTION_BLOCK Module_1_Virtualfunctionalblock
(******************************************)
(* Automatic generated code, do not edit! *)
(******************************************)
VAR_INPUT
	bObjectIndex : BYTE := 0;
	VT_Request1 : typSnvtObjRequest;
	VT_TimeSet1 : typSnvtTimeStamp;
	VT_AlarmSet1 : typSnvtAlarm;
	VT_DHW_ModeSet1 : typSnvtHvacMode;
	VT_DHW_SetPoint1 : typSnvtTempP;
	VT_CFD_SetEn1 : typSnvtSwitch;
	VT_CFD_SetMode1 : typSnvtHvacMode;
	VT_CFD_SetPoint1 : typSnvtTempP;
	VT_Request2 : typSnvtObjRequest;
	VT_TimeSet2 : typSnvtTimeStamp;
	VT_AlarmSet2 : typSnvtAlarm;
	VT_DHW_ModeSet2 : typSnvtHvacMode;
	VT_DHW_SetPoint2 : typSnvtTempP;
	VT_CFD_SetEn2 : typSnvtSwitch;
	VT_CFD_SetMode2 : typSnvtHvacMode;
	VT_CFD_SetPoint2 : typSnvtTempP;

END_VAR
VAR_OUTPUT
	VT_Status1 : typSnvtObjStatus;
	VT_Alarm1 : typSnvtAlarm;
	VT_RlyState1 : typSnvtState;
	VT_DHW_ActTemp1 : typSnvtTempP;
	VT_DHW_SetTemp1 : typSnvtTempP;
	VT_CFD_GetEn1 : typSnvtSwitch;
	VT_CFD_Temp1 : typSnvtTempP;
	VT_CFD_SetTemp1 : typSnvtTempP;
	VT_Status2 : typSnvtObjStatus;
	VT_Alarm2 : typSnvtAlarm;
	VT_RlyState2 : typSnvtState;
	VT_DHW_ActTemp2 : typSnvtTempP;
	VT_DHW_SetTemp2 : typSnvtTempP;
	VT_CFD_GetEn2 : typSnvtSwitch;
	VT_CFD_Temp2 : typSnvtTempP;
	VT_CFD_SetTemp2 : typSnvtTempP;

END_VAR
VAR
	xSetOnce : BOOL := TRUE;
	xDataInUpdated : BOOL := FALSE;
	paNviSnvtObjStatus : ARRAY[0..1] OF POINTER TO typSnvtObjStatus;
	aNviSnvtObjStatusIndex : ARRAY[0..1] OF BYTE := 1,17;
	paNviSnvtAlarm : ARRAY[0..1] OF POINTER TO typSnvtAlarm;
	aNviSnvtAlarmIndex : ARRAY[0..1] OF BYTE := 3,19;
	paNviSnvtState : ARRAY[0..1] OF POINTER TO typSnvtState;
	aNviSnvtStateIndex : ARRAY[0..1] OF BYTE := 5,21;
	paNviSnvtTempP : ARRAY[0..7] OF POINTER TO typSnvtTempP;
	aNviSnvtTempPIndex : ARRAY[0..7] OF BYTE := 7,9,13,15,23,25,29,31;
	paNviSnvtSwitch : ARRAY[0..1] OF POINTER TO typSnvtSwitch;
	aNviSnvtSwitchIndex : ARRAY[0..1] OF BYTE := 11,27;
	paNvoSnvtObjRequest : ARRAY[0..1] OF POINTER TO typSnvtObjRequest;
	aNvoSnvtObjRequestIndex : ARRAY[0..1] OF BYTE := 0,16;
	aNvoSnvtObjRequestLast : ARRAY[0..1] OF typSnvtObjRequest;
	aNvoSnvtObjRequestPriority : ARRAY[0..0] OF BYTE := 16#00;
	paNvoSnvtTimeStamp : ARRAY[0..1] OF POINTER TO typSnvtTimeStamp;
	aNvoSnvtTimeStampIndex : ARRAY[0..1] OF BYTE := 2,18;
	aNvoSnvtTimeStampLast : ARRAY[0..1] OF typSnvtTimeStamp;
	aNvoSnvtTimeStampPriority : ARRAY[0..0] OF BYTE := 16#00;
	paNvoSnvtAlarm : ARRAY[0..1] OF POINTER TO typSnvtAlarm;
	aNvoSnvtAlarmIndex : ARRAY[0..1] OF BYTE := 4,20;
	aNvoSnvtAlarmLast : ARRAY[0..1] OF typSnvtAlarm;
	aNvoSnvtAlarmPriority : ARRAY[0..0] OF BYTE := 16#00;
	paNvoSnvtHvacMode : ARRAY[0..3] OF POINTER TO typSnvtHvacMode;
	aNvoSnvtHvacModeIndex : ARRAY[0..3] OF BYTE := 6,12,22,28;
	aNvoSnvtHvacModeLast : ARRAY[0..3] OF typSnvtHvacMode;
	aNvoSnvtHvacModePriority : ARRAY[0..0] OF BYTE := 16#00;
	paNvoSnvtTempP : ARRAY[0..3] OF POINTER TO typSnvtTempP;
	aNvoSnvtTempPIndex : ARRAY[0..3] OF BYTE := 8,14,24,30;
	aNvoSnvtTempPLast : ARRAY[0..3] OF typSnvtTempP;
	aNvoSnvtTempPPriority : ARRAY[0..0] OF BYTE := 16#00;
	paNvoSnvtSwitch : ARRAY[0..1] OF POINTER TO typSnvtSwitch;
	aNvoSnvtSwitchIndex : ARRAY[0..1] OF BYTE := 10,26;
	aNvoSnvtSwitchLast : ARRAY[0..1] OF typSnvtSwitch;
	aNvoSnvtSwitchPriority : ARRAY[0..0] OF BYTE := 16#00;

	cmd : BYTE;
	z : INT;
	bNvRelativeIdx : BYTE;
	bNvAbsoluteIdx : BYTE;
	wCpRelativeIdx : WORD;
	wCpAbsoluteIdx : WORD;
END_VAR
VAR CONSTANT
	bNvStartIndex : BYTE := 5;
	wCpStartIndex : WORD := 65535;
	bLmoCount : BYTE := 1;
END_VAR
IF (xInitRunning_Module_1 = TRUE) AND (xSetOnce = TRUE) THEN
	xSetOnce := FALSE;
	CachePointers();
	SetUpdateFlags();
END_IF

CheckUpdateFlags();
IF (xInitRunning_Module_1 = FALSE) AND (xDataInUpdated = FALSE) THEN
	IF (mbxModule_1.bStatus.0) THEN
		SendValueRequest();
	END_IF
END_IF

IF (xInitRunning_Module_1 = FALSE) AND (mbxModule_1.bStatus.0) THEN
	xSetOnce := TRUE;
	xDataInUpdated := FALSE;
	FOR z := 0 TO 1 DO
		IF ((NOT FuMemCompare(ADR(aNvoSnvtObjRequestLast[z]), paNvoSnvtObjRequest[z], ADR(paNvoSnvtObjRequest[z]^.bStatusInformation) - paNvoSnvtObjRequest[z])) OR (paNvoSnvtObjRequest[z]^.bStatusInformation.7 = TRUE) OR (aNvoSnvtObjRequestLast[z].bInternalUseOnly.1 = TRUE)) THEN
			FuSnvtObjRequestToRaw(paNvoSnvtObjRequest[z], ADR(OutDataTelegram_Module_1[2]));

			bNvAbsoluteIdx := bNvStartIndex + bObjectIndex + (aNvoSnvtObjRequestIndex[z] * bLmoCount);

			IF (FuDoNvoUpdate_Module_1(paNvoSnvtObjRequest[z], ADR(aNvoSnvtObjRequestLast[z]), ADR(paNvoSnvtObjRequest[z]^.bInternalUseOnly), ADR(aNvoSnvtObjRequestLast[z].bInternalUseOnly), ADR(paNvoSnvtObjRequest[z]^.bStatusInformation), bNvAbsoluteIdx, 3, SIZEOF(aNvoSnvtObjRequestLast[z])) = FALSE) THEN
				RETURN;
			END_IF
		END_IF
	END_FOR
	FOR z := 0 TO 1 DO
		IF ((NOT FuMemCompare(ADR(aNvoSnvtTimeStampLast[z]), paNvoSnvtTimeStamp[z], ADR(paNvoSnvtTimeStamp[z]^.bStatusInformation) - paNvoSnvtTimeStamp[z])) OR (paNvoSnvtTimeStamp[z]^.bStatusInformation.7 = TRUE) OR (aNvoSnvtTimeStampLast[z].bInternalUseOnly.1 = TRUE)) THEN
			FuSnvtTimeStampToRaw(paNvoSnvtTimeStamp[z], ADR(OutDataTelegram_Module_1[2]));

			bNvAbsoluteIdx := bNvStartIndex + bObjectIndex + (aNvoSnvtTimeStampIndex[z] * bLmoCount);

			IF (FuDoNvoUpdate_Module_1(paNvoSnvtTimeStamp[z], ADR(aNvoSnvtTimeStampLast[z]), ADR(paNvoSnvtTimeStamp[z]^.bInternalUseOnly), ADR(aNvoSnvtTimeStampLast[z].bInternalUseOnly), ADR(paNvoSnvtTimeStamp[z]^.bStatusInformation), bNvAbsoluteIdx, 7, SIZEOF(aNvoSnvtTimeStampLast[z])) = FALSE) THEN
				RETURN;
			END_IF
		END_IF
	END_FOR
	FOR z := 0 TO 1 DO
		IF ((NOT FuMemCompare(ADR(aNvoSnvtAlarmLast[z]), paNvoSnvtAlarm[z], ADR(paNvoSnvtAlarm[z]^.bStatusInformation) - paNvoSnvtAlarm[z])) OR (paNvoSnvtAlarm[z]^.bStatusInformation.7 = TRUE) OR (aNvoSnvtAlarmLast[z].bInternalUseOnly.1 = TRUE)) THEN
			FuSnvtAlarmToRaw(paNvoSnvtAlarm[z], ADR(OutDataTelegram_Module_1[2]));

			bNvAbsoluteIdx := bNvStartIndex + bObjectIndex + (aNvoSnvtAlarmIndex[z] * bLmoCount);

			IF (FuDoNvoUpdate_Module_1(paNvoSnvtAlarm[z], ADR(aNvoSnvtAlarmLast[z]), ADR(paNvoSnvtAlarm[z]^.bInternalUseOnly), ADR(aNvoSnvtAlarmLast[z].bInternalUseOnly), ADR(paNvoSnvtAlarm[z]^.bStatusInformation), bNvAbsoluteIdx, 29, SIZEOF(aNvoSnvtAlarmLast[z])) = FALSE) THEN
				RETURN;
			END_IF
		END_IF
	END_FOR
	FOR z := 0 TO 3 DO
		IF ((NOT FuMemCompare(ADR(aNvoSnvtHvacModeLast[z]), paNvoSnvtHvacMode[z], ADR(paNvoSnvtHvacMode[z]^.bStatusInformation) - paNvoSnvtHvacMode[z])) OR (paNvoSnvtHvacMode[z]^.bStatusInformation.7 = TRUE) OR (aNvoSnvtHvacModeLast[z].bInternalUseOnly.1 = TRUE)) THEN
			FuSnvtHvacModeToRaw(paNvoSnvtHvacMode[z], ADR(OutDataTelegram_Module_1[2]));

			bNvAbsoluteIdx := bNvStartIndex + bObjectIndex + (aNvoSnvtHvacModeIndex[z] * bLmoCount);

			IF (FuDoNvoUpdate_Module_1(paNvoSnvtHvacMode[z], ADR(aNvoSnvtHvacModeLast[z]), ADR(paNvoSnvtHvacMode[z]^.bInternalUseOnly), ADR(aNvoSnvtHvacModeLast[z].bInternalUseOnly), ADR(paNvoSnvtHvacMode[z]^.bStatusInformation), bNvAbsoluteIdx, 1, SIZEOF(aNvoSnvtHvacModeLast[z])) = FALSE) THEN
				RETURN;
			END_IF
		END_IF
	END_FOR
	FOR z := 0 TO 3 DO
		IF ((NOT FuMemCompare(ADR(aNvoSnvtTempPLast[z]), paNvoSnvtTempP[z], ADR(paNvoSnvtTempP[z]^.bStatusInformation) - paNvoSnvtTempP[z])) OR (paNvoSnvtTempP[z]^.bStatusInformation.7 = TRUE) OR (aNvoSnvtTempPLast[z].bInternalUseOnly.1 = TRUE)) THEN
			FuSnvtTempPToRaw(paNvoSnvtTempP[z], ADR(OutDataTelegram_Module_1[2]));

			bNvAbsoluteIdx := bNvStartIndex + bObjectIndex + (aNvoSnvtTempPIndex[z] * bLmoCount);

			IF (FuDoNvoUpdate_Module_1(paNvoSnvtTempP[z], ADR(aNvoSnvtTempPLast[z]), ADR(paNvoSnvtTempP[z]^.bInternalUseOnly), ADR(aNvoSnvtTempPLast[z].bInternalUseOnly), ADR(paNvoSnvtTempP[z]^.bStatusInformation), bNvAbsoluteIdx, 2, SIZEOF(aNvoSnvtTempPLast[z])) = FALSE) THEN
				RETURN;
			END_IF
		END_IF
	END_FOR
	FOR z := 0 TO 1 DO
		IF ((NOT FuMemCompare(ADR(aNvoSnvtSwitchLast[z]), paNvoSnvtSwitch[z], ADR(paNvoSnvtSwitch[z]^.bStatusInformation) - paNvoSnvtSwitch[z])) OR (paNvoSnvtSwitch[z]^.bStatusInformation.7 = TRUE) OR (aNvoSnvtSwitchLast[z].bInternalUseOnly.1 = TRUE)) THEN
			FuSnvtSwitchToRaw(paNvoSnvtSwitch[z], ADR(OutDataTelegram_Module_1[2]));

			bNvAbsoluteIdx := bNvStartIndex + bObjectIndex + (aNvoSnvtSwitchIndex[z] * bLmoCount);

			IF (FuDoNvoUpdate_Module_1(paNvoSnvtSwitch[z], ADR(aNvoSnvtSwitchLast[z]), ADR(paNvoSnvtSwitch[z]^.bInternalUseOnly), ADR(aNvoSnvtSwitchLast[z].bInternalUseOnly), ADR(paNvoSnvtSwitch[z]^.bStatusInformation), bNvAbsoluteIdx, 2, SIZEOF(aNvoSnvtSwitchLast[z])) = FALSE) THEN
				RETURN;
			END_IF
		END_IF
	END_FOR

END_IF
END_FUNCTION_BLOCK
ACTION CachePointers:
paNviSnvtObjStatus[0] := ADR(VT_Status1);
paNviSnvtObjStatus[1] := ADR(VT_Status2);
paNviSnvtAlarm[0] := ADR(VT_Alarm1);
paNviSnvtAlarm[1] := ADR(VT_Alarm2);
paNviSnvtState[0] := ADR(VT_RlyState1);
paNviSnvtState[1] := ADR(VT_RlyState2);
paNviSnvtTempP[0] := ADR(VT_DHW_ActTemp1);
paNviSnvtTempP[1] := ADR(VT_DHW_SetTemp1);
paNviSnvtTempP[2] := ADR(VT_CFD_Temp1);
paNviSnvtTempP[3] := ADR(VT_CFD_SetTemp1);
paNviSnvtTempP[4] := ADR(VT_DHW_ActTemp2);
paNviSnvtTempP[5] := ADR(VT_DHW_SetTemp2);
paNviSnvtTempP[6] := ADR(VT_CFD_Temp2);
paNviSnvtTempP[7] := ADR(VT_CFD_SetTemp2);
paNviSnvtSwitch[0] := ADR(VT_CFD_GetEn1);
paNviSnvtSwitch[1] := ADR(VT_CFD_GetEn2);
paNvoSnvtObjRequest[0] := ADR(VT_Request1);
paNvoSnvtObjRequest[1] := ADR(VT_Request2);
paNvoSnvtTimeStamp[0] := ADR(VT_TimeSet1);
paNvoSnvtTimeStamp[1] := ADR(VT_TimeSet2);
paNvoSnvtAlarm[0] := ADR(VT_AlarmSet1);
paNvoSnvtAlarm[1] := ADR(VT_AlarmSet2);
paNvoSnvtHvacMode[0] := ADR(VT_DHW_ModeSet1);
paNvoSnvtHvacMode[1] := ADR(VT_CFD_SetMode1);
paNvoSnvtHvacMode[2] := ADR(VT_DHW_ModeSet2);
paNvoSnvtHvacMode[3] := ADR(VT_CFD_SetMode2);
paNvoSnvtTempP[0] := ADR(VT_DHW_SetPoint1);
paNvoSnvtTempP[1] := ADR(VT_CFD_SetPoint1);
paNvoSnvtTempP[2] := ADR(VT_DHW_SetPoint2);
paNvoSnvtTempP[3] := ADR(VT_CFD_SetPoint2);
paNvoSnvtSwitch[0] := ADR(VT_CFD_SetEn1);
paNvoSnvtSwitch[1] := ADR(VT_CFD_SetEn2);
;
END_ACTION
ACTION CheckUpdateFlags:
xDataInUpdated := TRUE;
FOR z := 0 TO 1 DO
	xDataInUpdated := xDataInUpdated AND (NOT paNviSnvtObjStatus[z]^.bInternalUseOnly.0);
END_FOR
FOR z := 0 TO 1 DO
	xDataInUpdated := xDataInUpdated AND (NOT paNviSnvtAlarm[z]^.bInternalUseOnly.0);
END_FOR
FOR z := 0 TO 1 DO
	xDataInUpdated := xDataInUpdated AND (NOT paNviSnvtState[z]^.bInternalUseOnly.0);
END_FOR
FOR z := 0 TO 7 DO
	xDataInUpdated := xDataInUpdated AND (NOT paNviSnvtTempP[z]^.bInternalUseOnly.0);
END_FOR
FOR z := 0 TO 1 DO
	xDataInUpdated := xDataInUpdated AND (NOT paNviSnvtSwitch[z]^.bInternalUseOnly.0);
END_FOR
END_ACTION
ACTION DataReceived:
cmd := InDataTelegram_Module_1[0];
IF (cmd = M2C_NVI_UPDT_OCCD) OR (cmd = M2C_NV_VALUE_RSP) OR (cmd = M2C_NVI_UPDT_TOUT) THEN
	bNvRelativeIdx := (InDataTelegram_Module_1[1] - bNvStartIndex - bObjectIndex) / bLmoCount;
	CASE bNvRelativeIdx OF
	1, 17:
		IF (cmd = M2C_NVI_UPDT_OCCD) OR (cmd = M2C_NV_VALUE_RSP) THEN
			IF (unLastLen_mbxModule_1 = (2 + 6)) THEN
				FOR z := 0 TO 1 DO
					IF aNviSnvtObjStatusIndex[z] = bNvRelativeIdx THEN
						FuRawToSnvtObjStatus(ADR(InDataTelegram_Module_1[2]), paNviSnvtObjStatus[z]);
						paNviSnvtObjStatus[z]^.bInternalUseOnly.0 := FALSE;
						paNviSnvtObjStatus[z]^.bStatusInformation := FuInkrementNviStatus(paNviSnvtObjStatus[z]^.bStatusInformation);
						EXIT;
					END_IF
				END_FOR
			ELSIF (unLastLen_mbxModule_1 = 2) THEN
				FOR z := 0 TO 1 DO
					IF aNviSnvtObjStatusIndex[z] = bNvRelativeIdx THEN
						paNviSnvtObjStatus[z]^.bStatusInformation := FuInkrementNviStatus(paNviSnvtObjStatus[z]^.bStatusInformation);
						EXIT;
					END_IF
				END_FOR
			END_IF
		ELSIF (cmd = M2C_NVI_UPDT_TOUT) THEN
			IF (unLastLen_mbxModule_1 = 3) THEN
				FOR z := 0 TO 1 DO
					IF aNviSnvtObjStatusIndex[z] = bNvRelativeIdx THEN
						paNviSnvtObjStatus[z]^.bStatusInformation.4 := BYTE_TO_BOOL(InDataTelegram_Module_1[2]);
						EXIT;
					END_IF
				END_FOR
			END_IF
		END_IF
	3, 19:
		IF (cmd = M2C_NVI_UPDT_OCCD) OR (cmd = M2C_NV_VALUE_RSP) THEN
			IF (unLastLen_mbxModule_1 = (2 + 29)) THEN
				FOR z := 0 TO 1 DO
					IF aNviSnvtAlarmIndex[z] = bNvRelativeIdx THEN
						FuRawToSnvtAlarm(ADR(InDataTelegram_Module_1[2]), paNviSnvtAlarm[z]);
						paNviSnvtAlarm[z]^.bInternalUseOnly.0 := FALSE;
						paNviSnvtAlarm[z]^.bStatusInformation := FuInkrementNviStatus(paNviSnvtAlarm[z]^.bStatusInformation);
						EXIT;
					END_IF
				END_FOR
			ELSIF (unLastLen_mbxModule_1 = 2) THEN
				FOR z := 0 TO 1 DO
					IF aNviSnvtAlarmIndex[z] = bNvRelativeIdx THEN
						paNviSnvtAlarm[z]^.bStatusInformation := FuInkrementNviStatus(paNviSnvtAlarm[z]^.bStatusInformation);
						EXIT;
					END_IF
				END_FOR
			END_IF
		ELSIF (cmd = M2C_NVI_UPDT_TOUT) THEN
			IF (unLastLen_mbxModule_1 = 3) THEN
				FOR z := 0 TO 1 DO
					IF aNviSnvtAlarmIndex[z] = bNvRelativeIdx THEN
						paNviSnvtAlarm[z]^.bStatusInformation.4 := BYTE_TO_BOOL(InDataTelegram_Module_1[2]);
						EXIT;
					END_IF
				END_FOR
			END_IF
		END_IF
	5, 21:
		IF (cmd = M2C_NVI_UPDT_OCCD) OR (cmd = M2C_NV_VALUE_RSP) THEN
			IF (unLastLen_mbxModule_1 = (2 + 2)) THEN
				FOR z := 0 TO 1 DO
					IF aNviSnvtStateIndex[z] = bNvRelativeIdx THEN
						FuRawToSnvtState(ADR(InDataTelegram_Module_1[2]), paNviSnvtState[z]);
						paNviSnvtState[z]^.bInternalUseOnly.0 := FALSE;
						paNviSnvtState[z]^.bStatusInformation := FuInkrementNviStatus(paNviSnvtState[z]^.bStatusInformation);
						EXIT;
					END_IF
				END_FOR
			ELSIF (unLastLen_mbxModule_1 = 2) THEN
				FOR z := 0 TO 1 DO
					IF aNviSnvtStateIndex[z] = bNvRelativeIdx THEN
						paNviSnvtState[z]^.bStatusInformation := FuInkrementNviStatus(paNviSnvtState[z]^.bStatusInformation);
						EXIT;
					END_IF
				END_FOR
			END_IF
		ELSIF (cmd = M2C_NVI_UPDT_TOUT) THEN
			IF (unLastLen_mbxModule_1 = 3) THEN
				FOR z := 0 TO 1 DO
					IF aNviSnvtStateIndex[z] = bNvRelativeIdx THEN
						paNviSnvtState[z]^.bStatusInformation.4 := BYTE_TO_BOOL(InDataTelegram_Module_1[2]);
						EXIT;
					END_IF
				END_FOR
			END_IF
		END_IF
	7, 9, 13, 15, 23, 25, 29, 31:
		IF (cmd = M2C_NVI_UPDT_OCCD) OR (cmd = M2C_NV_VALUE_RSP) THEN
			IF (unLastLen_mbxModule_1 = (2 + 2)) THEN
				FOR z := 0 TO 7 DO
					IF aNviSnvtTempPIndex[z] = bNvRelativeIdx THEN
						FuRawToSnvtTempP(ADR(InDataTelegram_Module_1[2]), paNviSnvtTempP[z]);
						paNviSnvtTempP[z]^.bInternalUseOnly.0 := FALSE;
						paNviSnvtTempP[z]^.bStatusInformation := FuInkrementNviStatus(paNviSnvtTempP[z]^.bStatusInformation);
						EXIT;
					END_IF
				END_FOR
			ELSIF (unLastLen_mbxModule_1 = 2) THEN
				FOR z := 0 TO 7 DO
					IF aNviSnvtTempPIndex[z] = bNvRelativeIdx THEN
						paNviSnvtTempP[z]^.bStatusInformation := FuInkrementNviStatus(paNviSnvtTempP[z]^.bStatusInformation);
						EXIT;
					END_IF
				END_FOR
			END_IF
		ELSIF (cmd = M2C_NVI_UPDT_TOUT) THEN
			IF (unLastLen_mbxModule_1 = 3) THEN
				FOR z := 0 TO 7 DO
					IF aNviSnvtTempPIndex[z] = bNvRelativeIdx THEN
						paNviSnvtTempP[z]^.bStatusInformation.4 := BYTE_TO_BOOL(InDataTelegram_Module_1[2]);
						EXIT;
					END_IF
				END_FOR
			END_IF
		END_IF
	11, 27:
		IF (cmd = M2C_NVI_UPDT_OCCD) OR (cmd = M2C_NV_VALUE_RSP) THEN
			IF (unLastLen_mbxModule_1 = (2 + 2)) THEN
				FOR z := 0 TO 1 DO
					IF aNviSnvtSwitchIndex[z] = bNvRelativeIdx THEN
						FuRawToSnvtSwitch(ADR(InDataTelegram_Module_1[2]), paNviSnvtSwitch[z]);
						paNviSnvtSwitch[z]^.bInternalUseOnly.0 := FALSE;
						paNviSnvtSwitch[z]^.bStatusInformation := FuInkrementNviStatus(paNviSnvtSwitch[z]^.bStatusInformation);
						EXIT;
					END_IF
				END_FOR
			ELSIF (unLastLen_mbxModule_1 = 2) THEN
				FOR z := 0 TO 1 DO
					IF aNviSnvtSwitchIndex[z] = bNvRelativeIdx THEN
						paNviSnvtSwitch[z]^.bStatusInformation := FuInkrementNviStatus(paNviSnvtSwitch[z]^.bStatusInformation);
						EXIT;
					END_IF
				END_FOR
			END_IF
		ELSIF (cmd = M2C_NVI_UPDT_TOUT) THEN
			IF (unLastLen_mbxModule_1 = 3) THEN
				FOR z := 0 TO 1 DO
					IF aNviSnvtSwitchIndex[z] = bNvRelativeIdx THEN
						paNviSnvtSwitch[z]^.bStatusInformation.4 := BYTE_TO_BOOL(InDataTelegram_Module_1[2]);
						EXIT;
					END_IF
				END_FOR
			END_IF
		END_IF

	END_CASE
ELSIF (cmd = M2C_CP_VALUE_RSP) THEN
	wCpRelativeIdx := ((InDataTelegram_Module_1[1] + InDataTelegram_Module_1[2] * 256) - wCpStartIndex - bObjectIndex) / bLmoCount;
	CASE wCpRelativeIdx OF

	END_CASE
END_IF
END_ACTION
ACTION ResetNviUpdate:
FOR z := 0 TO 1 DO
	paNviSnvtObjStatus[z]^.bStatusInformation := paNviSnvtObjStatus[z]^.bStatusInformation AND 16#F8;
END_FOR
FOR z := 0 TO 1 DO
	paNviSnvtAlarm[z]^.bStatusInformation := paNviSnvtAlarm[z]^.bStatusInformation AND 16#F8;
END_FOR
FOR z := 0 TO 1 DO
	paNviSnvtState[z]^.bStatusInformation := paNviSnvtState[z]^.bStatusInformation AND 16#F8;
END_FOR
FOR z := 0 TO 7 DO
	paNviSnvtTempP[z]^.bStatusInformation := paNviSnvtTempP[z]^.bStatusInformation AND 16#F8;
END_FOR
FOR z := 0 TO 1 DO
	paNviSnvtSwitch[z]^.bStatusInformation := paNviSnvtSwitch[z]^.bStatusInformation AND 16#F8;
END_FOR
;
END_ACTION
ACTION SendValueRequest:
FOR z := 0 TO 1 DO
	IF (FuSendNviValueReq_Module_1(ADR(paNviSnvtObjStatus[z]^.bInternalUseOnly), bNvStartIndex + bObjectIndex + (aNviSnvtObjStatusIndex[z] * bLmoCount)) = FALSE) THEN
		RETURN;
	END_IF;
END_FOR;
FOR z := 0 TO 1 DO
	IF (FuSendNviValueReq_Module_1(ADR(paNviSnvtAlarm[z]^.bInternalUseOnly), bNvStartIndex + bObjectIndex + (aNviSnvtAlarmIndex[z] * bLmoCount)) = FALSE) THEN
		RETURN;
	END_IF;
END_FOR;
FOR z := 0 TO 1 DO
	IF (FuSendNviValueReq_Module_1(ADR(paNviSnvtState[z]^.bInternalUseOnly), bNvStartIndex + bObjectIndex + (aNviSnvtStateIndex[z] * bLmoCount)) = FALSE) THEN
		RETURN;
	END_IF;
END_FOR;
FOR z := 0 TO 7 DO
	IF (FuSendNviValueReq_Module_1(ADR(paNviSnvtTempP[z]^.bInternalUseOnly), bNvStartIndex + bObjectIndex + (aNviSnvtTempPIndex[z] * bLmoCount)) = FALSE) THEN
		RETURN;
	END_IF;
END_FOR;
FOR z := 0 TO 1 DO
	IF (FuSendNviValueReq_Module_1(ADR(paNviSnvtSwitch[z]^.bInternalUseOnly), bNvStartIndex + bObjectIndex + (aNviSnvtSwitchIndex[z] * bLmoCount)) = FALSE) THEN
		RETURN;
	END_IF;
END_FOR;
;
END_ACTION
ACTION SetUpdateFlags:
FOR z := 0 TO 1 DO
	paNviSnvtObjStatus[z]^.bInternaluseOnly.0 := TRUE;
END_FOR;
FOR z := 0 TO 1 DO
	paNviSnvtAlarm[z]^.bInternaluseOnly.0 := TRUE;
END_FOR;
FOR z := 0 TO 1 DO
	paNviSnvtState[z]^.bInternaluseOnly.0 := TRUE;
END_FOR;
FOR z := 0 TO 7 DO
	paNviSnvtTempP[z]^.bInternaluseOnly.0 := TRUE;
END_FOR;
FOR z := 0 TO 1 DO
	paNviSnvtSwitch[z]^.bInternaluseOnly.0 := TRUE;
END_FOR;
FOR z := 0 TO 1 DO
	aNvoSnvtObjRequestLast[z].bInternaluseOnly.1 := TRUE;
	aNvoSnvtObjRequestLast[z].bInternaluseOnly.7 := (SHR(aNvoSnvtObjRequestPriority[z / 8], z MOD 8) AND 1) <> 0;
END_FOR;
FOR z := 0 TO 1 DO
	aNvoSnvtTimeStampLast[z].bInternaluseOnly.1 := TRUE;
	aNvoSnvtTimeStampLast[z].bInternaluseOnly.7 := (SHR(aNvoSnvtTimeStampPriority[z / 8], z MOD 8) AND 1) <> 0;
END_FOR;
FOR z := 0 TO 1 DO
	aNvoSnvtAlarmLast[z].bInternaluseOnly.1 := TRUE;
	aNvoSnvtAlarmLast[z].bInternaluseOnly.7 := (SHR(aNvoSnvtAlarmPriority[z / 8], z MOD 8) AND 1) <> 0;
END_FOR;
FOR z := 0 TO 3 DO
	aNvoSnvtHvacModeLast[z].bInternaluseOnly.1 := TRUE;
	aNvoSnvtHvacModeLast[z].bInternaluseOnly.7 := (SHR(aNvoSnvtHvacModePriority[z / 8], z MOD 8) AND 1) <> 0;
END_FOR;
FOR z := 0 TO 3 DO
	aNvoSnvtTempPLast[z].bInternaluseOnly.1 := TRUE;
	aNvoSnvtTempPLast[z].bInternaluseOnly.7 := (SHR(aNvoSnvtTempPPriority[z / 8], z MOD 8) AND 1) <> 0;
END_FOR;
FOR z := 0 TO 1 DO
	aNvoSnvtSwitchLast[z].bInternaluseOnly.1 := TRUE;
	aNvoSnvtSwitchLast[z].bInternaluseOnly.7 := (SHR(aNvoSnvtSwitchPriority[z / 8], z MOD 8) AND 1) <> 0;
END_FOR;
;
END_ACTION

(* POU LON/Shared/Internal/FuSnvtObjRequestToRaw, ST *)
FUNCTION FuSnvtObjRequestToRaw : BOOL
(******************************************)
(* Automatic generated code, do not edit! *)
(******************************************)
VAR_INPUT
	NvDataIn :  POINTER TO typSnvtObjRequest;
	DataOut : POINTER TO ARRAY[0..2] OF BYTE;
END_VAR
VAR
END_VAR
DataOut^[0] := WORD_TO_BYTE(SHR(NvDataIn^.wObjectId, 8));
DataOut^[1] := WORD_TO_BYTE(NvDataIn^.wObjectId);

DataOut^[2] := NvDataIn^.bObjectRequest;

FuSnvtObjRequestToRaw := TRUE;
END_FUNCTION

(* POU LON/Shared/Internal/FuSnvtTimeStampToRaw, ST *)
FUNCTION FuSnvtTimeStampToRaw : BOOL
(******************************************)
(* Automatic generated code, do not edit! *)
(******************************************)
VAR_INPUT
	NvDataIn :  POINTER TO typSnvtTimeStamp;
	DataOut : POINTER TO ARRAY[0..6] OF BYTE;
END_VAR
VAR
END_VAR
DataOut^[0] := INT_TO_BYTE(SHR(NvDataIn^.iYear, 8));
DataOut^[1] := INT_TO_BYTE(NvDataIn^.iYear);

DataOut^[2] := NvDataIn^.bMonth;

DataOut^[3] := NvDataIn^.bDay;

DataOut^[4] := NvDataIn^.bHour;

DataOut^[5] := NvDataIn^.bMinute;

DataOut^[6] := NvDataIn^.bSecond;

FuSnvtTimeStampToRaw := TRUE;
END_FUNCTION

(* POU LON/Shared/Internal/FuSnvtAlarmToRaw, ST *)
FUNCTION FuSnvtAlarmToRaw : BOOL
(******************************************)
(* Automatic generated code, do not edit! *)
(******************************************)
VAR_INPUT
	NvDataIn :  POINTER TO typSnvtAlarm;
	DataOut : POINTER TO ARRAY[0..28] OF BYTE;
END_VAR
VAR
END_VAR
DataOut^[0] := NvDataIn^.abLocation[0];
DataOut^[1] := NvDataIn^.abLocation[1];
DataOut^[2] := NvDataIn^.abLocation[2];
DataOut^[3] := NvDataIn^.abLocation[3];
DataOut^[4] := NvDataIn^.abLocation[4];
DataOut^[5] := NvDataIn^.abLocation[5];

DataOut^[6] := WORD_TO_BYTE(SHR(NvDataIn^.wObjectId, 8));
DataOut^[7] := WORD_TO_BYTE(NvDataIn^.wObjectId);

DataOut^[8] := NvDataIn^.bAlarmType;

DataOut^[9] := NvDataIn^.bPriorityLevel;

DataOut^[10] := WORD_TO_BYTE(SHR(NvDataIn^.wIndexToSnvt, 8));
DataOut^[11] := WORD_TO_BYTE(NvDataIn^.wIndexToSnvt);

DataOut^[12] := NvDataIn^.abValue[0];
DataOut^[13] := NvDataIn^.abValue[1];
DataOut^[14] := NvDataIn^.abValue[2];
DataOut^[15] := NvDataIn^.abValue[3];

DataOut^[16] := WORD_TO_BYTE(SHR(NvDataIn^.wYear, 8));
DataOut^[17] := WORD_TO_BYTE(NvDataIn^.wYear);

DataOut^[18] := NvDataIn^.bMonth;

DataOut^[19] := NvDataIn^.bDay;

DataOut^[20] := NvDataIn^.bHour;

DataOut^[21] := NvDataIn^.bMinute;

DataOut^[22] := NvDataIn^.bSecond;

DataOut^[23] := WORD_TO_BYTE(SHR(NvDataIn^.wMillisecond, 8));
DataOut^[24] := WORD_TO_BYTE(NvDataIn^.wMillisecond);

DataOut^[25] := NvDataIn^.abAlarmLimit[0];
DataOut^[26] := NvDataIn^.abAlarmLimit[1];
DataOut^[27] := NvDataIn^.abAlarmLimit[2];
DataOut^[28] := NvDataIn^.abAlarmLimit[3];

FuSnvtAlarmToRaw := TRUE;
END_FUNCTION

(* POU LON/Shared/Internal/FuSnvtHvacModeToRaw, ST *)
FUNCTION FuSnvtHvacModeToRaw : BOOL
(******************************************)
(* Automatic generated code, do not edit! *)
(******************************************)
VAR_INPUT
	NvDataIn :  POINTER TO typSnvtHvacMode;
	DataOut : POINTER TO ARRAY[0..0] OF BYTE;
END_VAR
VAR
END_VAR
DataOut^[0] := NvDataIn^.bSnvtHvacMode;

FuSnvtHvacModeToRaw := TRUE;
END_FUNCTION

(* POU LON/Shared/Internal/FuSnvtTempPToRaw, ST *)
FUNCTION FuSnvtTempPToRaw : BOOL
(******************************************)
(* Automatic generated code, do not edit! *)
(******************************************)
VAR_INPUT
	NvDataIn :  POINTER TO typSnvtTempP;
	DataOut : POINTER TO ARRAY[0..1] OF BYTE;
END_VAR
VAR
END_VAR
DataOut^[0] := INT_TO_BYTE(SHR(NvDataIn^.iSnvtTempP, 8));
DataOut^[1] := INT_TO_BYTE(NvDataIn^.iSnvtTempP);

FuSnvtTempPToRaw := TRUE;
END_FUNCTION

(* POU LON/Shared/Internal/FuSnvtSwitchToRaw, ST *)
FUNCTION FuSnvtSwitchToRaw : BOOL
(******************************************)
(* Automatic generated code, do not edit! *)
(******************************************)
VAR_INPUT
	NvDataIn :  POINTER TO typSnvtSwitch;
	DataOut : POINTER TO ARRAY[0..1] OF BYTE;
END_VAR
VAR
END_VAR
DataOut^[0] := NvDataIn^.bValue;

DataOut^[1] := NvDataIn^.siState;

FuSnvtSwitchToRaw := TRUE;
END_FUNCTION

(* POU TCP_Logger/Logger_Proc, ST *)
PROGRAM Logger_Proc
VAR
	c1:         	TCPCLIENT;

	Open:	    	BOOL;
	IpAddr:			DWORD;
	InetAddr:		DWORD;
	Connected:  	BOOL;
	Error:      	DINT;
	TxTrig:     	BOOL;
	RxData:			ARRAY [0..MAX_RECEIVE_TCP_CLIENT] OF BYTE;
	RxLen:			DINT;

	Retry:			BYTE;	(* Counter for connection retries *)
	Recovered:		BYTE;	(* Counter for recovered unsent messages *)

	i:				DINT;
	pos:			DWORD;
	hFile:			DWORD;

END_VAR
(*=== State machine ===*)
CASE Logger.Status OF

	S_Logger_UNKNOWN:
		(* Startup *)
		Logger.SendReq:=FALSE;
		Open:=FALSE;
		Logger.Status:=S_Logger_IDLE;

	S_Logger_IDLE:
		(* Wait request *)
		IF Logger.SendReq THEN
			(* Resolve server name or use static IP *)
			IF LEN(Logger_SERVER)=0 THEN
				InetAddr:=SysSockInetAddr(Logger_IP);
			ELSE
				IpAddr:=SysSockGetHostByName(ADR(Logger_SERVER));
				DWORDSWAP(pIn:=ADR(IpAddr), pOut:=ADR(InetAddr));
			END_IF
			TxTrig:=FALSE;
			RxLen:=0;
			(* Open connection *)
			Open:=TRUE;
			Logger.Status:=S_Logger_WAITCONN;
		END_IF

	S_Logger_WAITCONN:
		(* Wait connection *)
		IF Connected THEN
			(* Send data *)
			TxTrig:=TRUE;
			Logger.Status:=S_Logger_WAITTX;
		END_IF
		IF Error>0 THEN
			Open:=FALSE;
			Logger.Status:=S_Logger_ERROR;
		END_IF

	S_Logger_WAITTX:
		(* Wait transmission *)
		IF NOT TxTrig THEN
			Logger.Status:=S_Logger_WAITRESP;
		END_IF
		IF Error>0 THEN
			Open:=FALSE;
			Logger.Status:=S_Logger_ERROR;
		END_IF

	S_Logger_WAITRESP:
		(* Wait response *)
		IF Connected=FALSE (* OR TIMEOUT!! *) THEN
			Open:=FALSE;
			(* Check response *)
			IF RxLen>=4 AND CHKSTRING(pString:=ADR(RxData), pPattern:=ADR(Logger_CHECK)) THEN
				Logger.SendReq:=FALSE;
				Retry:=0;
				(* Check unsent messages to flush *)
				IF Recovered<Logger_RecoverMsgs THEN
					MsgChk();
					IF Logger.SendReq=TRUE THEN
						Recovered:=Recovered+1;
					ELSE
						Recovered:=0;
					END_IF
				ELSE
					Recovered:=0;
				END_IF
				Logger.Status:=S_Logger_IDLE;
			ELSE
				Logger.Status:=S_Logger_ERROR;
			END_IF
		END_IF

	S_Logger_ERROR:
		(* Connection error or send failure *)
		Retry:=Retry+1;
		IF Retry>Logger_ConnRetries THEN
			(* Save message as unsent *)
			MsgSave();
			Logger.SendReq:=FALSE;
			Retry:=0;
		END_IF
		Logger.Status:=S_Logger_IDLE;

ELSE
	Logger.Status:=S_Logger_UNKNOWN;
END_CASE


(*=== Execute client lib ===*)
c1(
	xOpenConnection			:= Open,
	dwInetAddr 				:= InetAddr,
	wPortNumber				:= Logger_PORT,
	ptSendData				:= ADR(Logger.SendData),
	diSendCount				:= Logger.SendLen,
	tConnectWatchdogTime	:= t#10s,
	xStartSend				:= TxTrig,
	aReceiveBuffer			:= RxData,
	diReceiveCount			:= RxLen,
	xConnected				=> Connected,
	diError					=> Error
);

(*=== Process Rx data ===*)
(*IF RxLen>0 THEN
	RxLen:=0;
END_IF*)
END_PROGRAM
ACTION MsgChk:
(* Open index file *)
hFile:=SysFileOpen(Logger_IndexFile,'r');
IF hFile=0 THEN
	RETURN;
END_IF
(* Search oldest message to recover *)
SysFileSetPos(hFile,Logger.LastIdxPos);
Logger.SendLen:=0;
REPEAT
	SysFileRead(hFile, ADR(Logger.SendIdx), SIZEOF(Logger.SendIdx));
	pos:=SysFileGetPos(hFile);
	SysFileRead(hFile, ADR(Logger.SendLen), SIZEOF(Logger.SendLen));
UNTIL
	SysFileEOF(hFile) OR Logger.SendLen<>0
END_REPEAT
SysFileClose(hFile);
(* Delete index file when all messages are recovered *)
IF Logger.SendLen=0 THEN
	Logger.LastIdxPos:=0;
	SysFileDelete(Logger_IndexFile);
	RETURN;
END_IF
(* Recover message data *)
hFile:=SysFileOpen(Logger_DataFile,'r');
IF hFile<>0 THEN
	SysFileSetPos(hFile,Logger.SendIdx);
	SysFileRead(hFile,ADR(Logger.SendData),Logger.SendLen);
	Logger.SendReq:=TRUE;
	SysFileClose(hFile);
END_IF
(* Clear index entry *)
hFile:=SysFileOpen(Logger_IndexFile,'a');
IF hFile<>0 THEN
	SysFileSetPos(hFile,pos);
	i:=0;
	SysFileWrite(hFile, ADR(i), 4);
	Logger.LastIdxPos:=SysFileGetPos(hFile);
	SysFileClose(hFile);
END_IF
END_ACTION
ACTION MsgSave:
(* Add log position in recovery indexes *)
hFile:=SysFileOpen(Logger_IndexFile,'a');
SysFileWrite(hFile, ADR(Logger.SendIdx), SIZEOF(Logger.SendIdx));
SysFileWrite(hFile, ADR(Logger.SendLen), SIZEOF(Logger.SendLen));
SysFileClose(hFile);
END_ACTION

